(* ---------------------------------------------------------------------------
Func name   : 	Off
Description : 	Sets the Indicator output to FALSE.
Inputs      :	None
Returns     : 	None
Notes       : 	
--------------------------------------------------------------------------- *)

METHOD Off
VAR_INPUT
END_VAR
m_signal^ := FALSE;
END_METHOD

(* ---------------------------------------------------------------------------
Func name   : 	On
Description : 	Sets the Indicator output to TRUE.
Inputs      :	None
Returns     : 	None
Notes       : 	
--------------------------------------------------------------------------- *)

METHOD On
VAR_INPUT
END_VAR
m_signal^ := TRUE;
END_METHOD

END_FUNCTION_BLOCK

// 20 Program Organization Units/Instrument-Controller Functions/fb_STARTP_ControlActuator
(*UPDATE: 			October. 29 2020 - Graham Hunter
					This function block converts a Real Signal/Command to a 4-20 mA signal to be processed by fb_AnalogOutputActuator.
					(Most of the functionality was duplicated from fb_ENDP_Analog but instead of converting a 4-20 mA signal to a Physical Signal, it converts a Physical Signal/Command to a 4-20 mA signal.)
*)

(*UPDATE: 			March. 18 2021 - Jaison Schaab

					Code Ported from Wago.
					
					Code has NOT Yet been tested.
*)

FUNCTION_BLOCK fb_STARTP_ControlActuator
VAR_INPUT
	PhysicalSignal 		: REAL; // this is a physical signal like speed
END_VAR
VAR_OUTPUT
	AnalogSignalValue   : REAL; // this is a 4-20 mA signal
	endpState : INT;
END_VAR
VAR
	m_pActuator420 : POINTER TO fb_AnalogOutputActuator;
	m_inMin 	: REAL;
	m_inMax 	: REAL;
	m_outMin 	: REAL;
	m_outMax 	: REAL;
	m_outpdiffMultiplier 	: REAL;
	m_inpdiffDivisor 		: REAL;
	m_offset 		: REAL;
	m_hysteresis 	: REAL;
	//this is all alarm-related down from here. Should be separated into Alarmable interface, if possible.
	m_devId					: UDeviceId;			// Device Id used for alarm integration
	//m_pAlarmHandler : POINTER TO fb_AlarmHandler; //Alarm handler function pointer
	LowAlarmMonitor 		: fb_AlarmMonitor;
	LowWarningMonitor 		: fb_AlarmMonitor;
	HighWarningMonitor 		: fb_AlarmMonitor;
	HighAlarmMonitor 		: fb_AlarmMonitor;
END_VAR
VAR CONSTANT
	DELAY_TON	: TIME := T#200MS;	//AlarmMonitor delay for Value to DEFINITEVILY cross the alarm limit boundary. and then Trigger.
END_VAR

//get transducers Value scaled from Physical to 4-20 
AnalogSignalValue := Scale(PhysicalSignal);

// None of the below is used currently on the 750-563 card currently <GRAHAM>
//Monitor alarms.
//LowAlarmMonitor.MonitorReal(AnalogSignalValue);
//LowWarningMonitor.MonitorReal(AnalogSignalValue);
//HighWarningMonitor.MonitorReal(AnalogSignalValue);
//HighAlarmMonitor.MonitorReal(AnalogSignalValue);

//ALSO_ update the so-called GaugeState. It controls Needle-Color. BY-DESIGN HW-Error also paints Needle in RED.

(* ---------------------------------------------------------------------------
Func name   : 	FB_init
Description : 	ENDP_Analog_Actuator
Inputs      :	4 reals - Two real values are the input range of the Physical Signal and Two real values are the output range of the Analog Signal.  
Returns     : 	None
--------------------------------------------------------------------------- *)

METHOD FB_init : BOOL
VAR_INPUT
	bInitRetains 		: BOOL; 		// if TRUE, the retain variables are initialized (warm start / cold start)
    bInCopyCode  		: BOOL; 		// if TRUE, the instance afterwards gets moved into the copy code (online change)
	
	//ptrActuator : POINTER TO fb_AnalogOutputActuator;
	PhysicalMin	: REAL;
	PhysicalMax	: REAL;
	AnalogMin 	: REAL;
	AnalogMax 	: REAL;
	//perctHysteresis : REAL;
END_VAR
//m_pActuator420 := ptrActuator;
m_inMin := PhysicalMin;
m_inMax := PhysicalMax;
m_outMin := AnalogMin;   //these are the range of analog values, 4-20 mA 0-10 VDC etc.
m_outMax := AnalogMax;    //that the physical signal is scaled to.
//m_outMin := m_pActuator420^.GetMinInput;   //these are the range of analog values, 4-20 mA 0-10 VDC etc.
//m_outMax := m_pActuator420^.GetMaxInput;    //that the physical signal is scaled to.
m_outpdiffMultiplier := (m_outMax - m_outMin);
m_inpdiffDivisor := (m_inMax - m_inMin);
IF (0.0 = m_inpdiffDivisor) THEN
	m_inpdiffDivisor := 0.000001; //protect against div-by-0, only ONCE, and produce VERY-LARGE Bad value.
                                  //Beckhoff-tcNov was doing this A.every cycle and B.returned 0.0 if Bad, which is normal value. hard to notice.
END_IF

//m_pAlarmHandler := ADR(gAlarmHandler); //i am no longer handling Alarms myself. AlarmMonitor does interfacing to 'gAlarmHandler'.
//m_devId := m_pTxducer420^.GetDevId();

//m_hysteresis := perctHysteresis/100;
//LowAlarmMonitor.Init(f_AlarmCode(m_devId, f_FaultCode(TFaultPriority.Warning, TFaultCondition.UnderLimit)), TAlarmMonitorType.lower_limit, DELAY_TON);
//LowWarningMonitor.Init(f_AlarmCode(m_devId, f_FaultCode(TFaultPriority.Warning, TFaultCondition.UnderWarning)), TAlarmMonitorType.lower_limit, DELAY_TON);
//HighWarningMonitor.Init(f_AlarmCode(m_devId, f_FaultCode(TFaultPriority.Warning, TFaultCondition.OverWarning)), TAlarmMonitorType.upper_limit, DELAY_TON);
//HighAlarmMonitor.Init(f_AlarmCode(m_devId, f_FaultCode(TFaultPriority.Warning, TFaultCondition.OverLimit)), TAlarmMonitorType.upper_limit, DELAY_TON);
END_METHOD

(* ---------------------------------------------------------------------------
Func name   : 	GetConfigData
Description : 	equivalent of "Configure" bkhff-legacy-names.
				
Inputs      :	2-end-range-values, 1 offset, 4 alarms - 7 values.
				state	-	state of the fault
Returns     : 	None
Notes       : 	
--------------------------------------------------------------------------- *)

METHOD GetConfigData
VAR_INPUT
	//cfg : TEndpAnalogCfg;
MinValue : REAL;
MaxValue : REAL;
OffsetValue : REAL;
END_VAR
m_outMin := MinValue;
m_outMax := MaxValue;
m_offset := OffsetValue;
END_METHOD

METHOD GetRange_MinMax
VAR_OUTPUT
	outMinVal : REAL;
	outMaxVal : REAL;
END_VAR
// these are the STARTP product values, in ANALOG UNITS
outMinVal := m_outMin;
outMaxVal := m_outMax;
END_METHOD

METHOD Scale : REAL
VAR_INPUT
	val_mamp : REAL;
END_VAR
Scale := (val_mamp - m_inMin)*m_outpdiffMultiplier/m_inpdiffDivisor + m_outMin;
END_METHOD

METHOD Set_Hysteresis
VAR_INPUT
	perctHysteresis : REAL;
END_VAR
m_hysteresis := perctHysteresis/100;
END_METHOD

METHOD SetRange_MinMax
VAR_INPUT
	AnalogMin : REAL;
	AnalogMax : REAL;
END_VAR
// these are the STARTP product values, in ANALOG Units <GRAHAM>
m_outMin := AnalogMin;
m_outMax := AnalogMax;
END_METHOD

END_FUNCTION_BLOCK

// 20 Program Organization Units/Instrument-Controller Functions/fb_Switch
(*AUTHOR:			Jaison Schaab*)
(*DATE:				March 27 / 2020*)
(*DESCRIPTION: 		This Function Block provides a standard conrol interface for digital
					inputs of type BOOL which includes a debounce feature.*)

(*UPDATE: 			March. 23 2021 - Jaison Schaab

					Code Is fully tested and functional.				
*)

(*UPDATE: 			March. 18 2021 - Jaison Schaab

					Code Ported from Wago.
					
					Code has NOT Yet been tested.
*)

(*UPDATE: 			September. 22 2020 - Jaison Schaab

					Updated the Equals routine to use a bistable block and second falling
					edge timer to now delay the falling edge of the input signal as well
					as the rising edge.
*)	

FUNCTION_BLOCK fb_Switch
VAR_INPUT
END_VAR
VAR_OUTPUT
END_VAR
VAR
	m_pSignal			: POINTER TO BOOL;	// Pointer to the input BOOL signal value
	m_debounce			: TIME;				// Debounce TIME value used for FALSE -> TRUE transition
	m_risingDelayTimer	: TON;				// Debounce timer used for FALSE -> TRUE transition
	m_fallingDelayTimer	: TON;				// Debounce timer used for TRUE -> FALSE transition
	m_signal			: RS;				// Output signal bistable block
END_VAR

(* ---------------------------------------------------------------------------
Func name   : 	Equals
Description : 	Retrieves the current switch value.
Inputs      :	None
Returns     : 	None
Notes       : 	This block is meant to be called cyclically to obtain the
				debounced value, there is no way to override operators in ST.
				
				The signal is delayed on both a FALSE -> TRUE transition
				and a TRUE -> FALSE transition.
--------------------------------------------------------------------------- *)

METHOD Equals : BOOL
VAR_INPUT
END_VAR
// use a rising edge delay timer to debounce the signal on a FALSE -> TRUE transition
m_risingDelayTimer(IN:= m_pSignal^, PT:= m_debounce, Q=> );

// use a falling edge delay timer to debounce the signal on a TRUE -> FALSE transition
m_fallingDelayTimer(IN:= NOT m_pSignal^, PT:= m_debounce, Q=> );

// Output the signal value
m_signal(SET:= m_risingDelayTimer.Q, RESET1:= m_fallingDelayTimer.Q, Q1=> Equals);
END_METHOD

(* ---------------------------------------------------------------------------
Func name   : 	FB_exit
Description : 	Destructor
Inputs      :	None
Returns     : 	None
Notes       : 	
--------------------------------------------------------------------------- *)

METHOD FB_exit : BOOL
VAR_INPUT
	bInCopyCode : BOOL; // if TRUE, the exit method is called for exiting an instance that is copied afterwards (online change)
END_VAR
// Do Nothing
END_METHOD

(* ---------------------------------------------------------------------------
Func name   : 	FB_init
Description : 	Constructor
Inputs      :	signal		-	Pointer to the input BOOL signal value
				debounce	-	Default debounce value of type TIME
Returns     : 	None
Notes       : 	
--------------------------------------------------------------------------- *)

METHOD FB_init : BOOL
VAR_INPUT
	bInitRetains 		: BOOL; 			// if TRUE, the retain variables are initialized (warm start / cold start)
    bInCopyCode  		: BOOL; 			// if TRUE, the instance afterwards gets moved into the copy code (online change)
	signal				: POINTER TO BOOL;	// Pointer to input BOOL signal value 
	debounce			: TIME := T#100MS;	// Default debounce value, can be overridden with Set routine
END_VAR
// Set the local signal pointer
m_pSignal := signal;

// Set the local debounce value to the default value
m_debounce := debounce;
END_METHOD

(* ---------------------------------------------------------------------------
Func name   : 	GetDebounce
Description : 	Gets the debounce time for the switch used to delay the
				the FALSE -> TRUE transition.
Inputs      :	None
Returns     : 	TIME	-	debounce TIME value
Notes       : 	
--------------------------------------------------------------------------- *)

METHOD GetDebounce : TIME
VAR_INPUT
END_VAR
GetDebounce := m_debounce;
END_METHOD

(* ---------------------------------------------------------------------------
Func name   : 	SetDebounce
Description : 	Sets the debounce time for the switch used to delay the
				the FALSE -> TRUE transition.
Inputs      :	debounce	- 	debounce TIME value
Returns     : 	None
Notes       : 	
--------------------------------------------------------------------------- *)

METHOD SetDebounce
VAR_INPUT
	debounce	: TIME;
END_VAR
m_debounce := debounce;
END_METHOD

END_FUNCTION_BLOCK

// 20 Program Organization Units/Interlock Functions/fb_NOVInterlock
(*AUTHOR:		Graham Hunter *)
(*DATE:			Feb 4, 2021 *)
(*DESCRIPTION:	Interlock logic block which interfaces with the NOV and NSA safety interlock PLC*)

(*NOTES:  

INPUTS: 	   Interface consists of external 13 interlock bit inputs and 15 interlock bit cmd override inputs (13 individual interlock override bits, one bypass All override bit, 
			   and one Bypass None Override bit). The Bypass All override supersedes all individual interlock bit overrides as well as the Bypass None override. 
			   The Bypass None override supersedes the individual interlock bit overrides. 
					
VAR_IN_OUTs:   The Function block takes in a VAR_IN_OUT process data structure of the THMINOVInterlock type (from the HMI) that consists of a interlock bit override input WORD (future use) 
			   as well as processed interlock bit output WORD.  
					
FUNCTIONALITY: This function block takes raw external individual interlock bit as inputs and with external individual override bits where one can override single individual interlock bits  
			   or bypass all the individual interlock bits or none of them. The override functionality can be done by the VAR_IN_OUT process data structure as well (in future use).
			   The seperate Process interlock Output word (in future use) will have the status for the individual processed interlock bits as well as status for the overall interlock with bypasses activated or 
			   bypasses not activated.
				  
OUTPUTS:      The output consists of individual processed interlock bits as well as overall status of the interlock block consisting of one ProcessedIntlkOK with No Bypasses bit and one
			  ProcessedIntlkOK with Bypasses. These output bits are fed into the VAR_IN_OUT process data structure.
	  
SIDE NOTE: 
			 Individual processed interlocks are TRUE = (INTLK IS TRUE OR OVERRIDE IS TRUE IF INDIVIDUAL OVERRIDE IS ACTIVE OR BYPASS ALL IS ACTIVE, 
												 FALSE = (INTLK IS FALSE AND OVERRIDE IS FALSE IF INDIVIDUAL OVERRIDE IS INACTIVE OR BYPASS ALL IS INACTIVE)
													
			 IF BYPASS NONE IS ACTIVE & BYPASS ALL IS INACTIVE then     
					processed interlocks are TRUE = (INTLK IS TRUE) 
											 FALSE = (INTLK IS FALSE)
			Note, BYPASS ALL Supersedes BYPASS NONE.
				
EXAMPLE CASE: If one has 3 interlocks out of the 13 used then set the other 10 non-used interlock bits to TRUE and the non-used overrides to FALSE (initially always set to FALSE). 
			  The Bypass All and Bypass None inputs commands can be used on the control engineers discretion.		
	*)
	
(* UPDATE:		April 22, 2021 - Graham Hunter

				Commented out a portion of the Interlock Processing code to be able to mimic NSA interlock logic where m_ProcessedIntlkOKWithBypass is True 
				with just the interlocks being satisfied without any overrides.
				
				Uncommented out the InitAlarms Method that initialize the alarms for when m_ProcessedIntlkOKWithBypass goes from True to False.
				Commented out the m_InterlocksOKAlarm.MonitorBool(value:= m_ProcessedIntlkOKWithBypass) code in fb_NOVInterlock. This code is not passed up as an output yet.
*)

FUNCTION_BLOCK fb_NOVInterlock
VAR_INPUT
	xEnable							: BOOL;
	//stInputData					: TNOVInterlockIn; // Not used as a seperate input from a external device currently, for future use <GRAHAM>
	Intlk01							: BOOL;	// TRUE = (INTLK SATISFIED), FALSE = (INTLK NOT SATISFIED)
	Intlk02							: BOOL;	
	Intlk03							: BOOL;	
	Intlk04							: BOOL;	
	Intlk05							: BOOL;	
	Intlk06							: BOOL;	
	Intlk07							: BOOL;	
	Intlk08							: BOOL;	
	Intlk09							: BOOL;	
	Intlk10							: BOOL;	
	Intlk11 						: BOOL;	
	Intlk12							: BOOL;	
	Intlk13							: BOOL;

	IntlkBypassALL					: BOOL;	// Bypass/override all interlocks command input
	Intlk01Bypass					: BOOL;	// TRUE = (OVERRIDE ACTIVE), FALSE = (OVERRIDE NOT ACTIVE)
	Intlk02Bypass					: BOOL;	
	Intlk03Bypass					: BOOL;	
	Intlk04Bypass					: BOOL;	
	Intlk05Bypass					: BOOL;	
	Intlk06Bypass					: BOOL;	
	Intlk07Bypass					: BOOL;	
	Intlk08Bypass					: BOOL;	
	Intlk09Bypass					: BOOL;	
	Intlk10Bypass					: BOOL;	
	Intlk11Bypass 					: BOOL;	
	Intlk12Bypass					: BOOL;	
	Intlk13Bypass					: BOOL;
	IntlkBypassNONE					: BOOL;	// Do not Bypass/override any interlocks command input	
END_VAR
VAR_OUTPUT
	//stOutputData					: TNOVInterlockStatusOut; // Possible future use of a seperate output WORD
	ProcessedIntlkOK_NoBypass		: BOOL;	// All interlocks are Ok with no bypasses/overrides
	ProcessedIntlk01				: BOOL;	// TRUE = (INTLK IS TRUE OR OVERRIDE IS TRUE IF OVERRIDE IS ACTIVE, FALSE = (INTLK IS FALSE AND OVERRIDE IS FALSE IF OVERRIDE IS ACTIVE)
	ProcessedIntlk02				: BOOL;	
	ProcessedIntlk03				: BOOL;	
	ProcessedIntlk04				: BOOL;	
	ProcessedIntlk05				: BOOL;	
	ProcessedIntlk06				: BOOL;	
	ProcessedIntlk07				: BOOL;	
	ProcessedIntlk08				: BOOL;	
	ProcessedIntlk09				: BOOL;	
	ProcessedIntlk10				: BOOL;	
	ProcessedIntlk11 				: BOOL;	
	ProcessedIntlk12				: BOOL;	
	ProcessedIntlk13				: BOOL;	
	ProcessedIntlkOK_WithBypass		: BOOL;	// All interlocks are Ok with bypasses/overrides
END_VAR
VAR_IN_OUT
	stProcessData					: THMINOVInterlock;	// Possible future use of a DynIn Bypass Cmd status input word
							
END_VAR

VAR
	
// Internal variables
// Internal Inputs
	// Interlock Status
	// Raw Unprocessed Interlocks from NOV or NSA interlocks 
	m_StatusIntlk01				: BOOL;					// TRUE = (INTLK SATISFIED), FALSE = (INTLK NOT SATISFIED)
	m_StatusIntlk02				: BOOL;					// TRUE = (INTLK SATISFIED), FALSE = (INTLK NOT SATISFIED)
	m_StatusIntlk03				: BOOL;					// TRUE = (INTLK SATISFIED), FALSE = (INTLK NOT SATISFIED)
	m_StatusIntlk04				: BOOL;					// TRUE = (INTLK SATISFIED), FALSE = (INTLK NOT SATISFIED)
	m_StatusIntlk05				: BOOL;					// TRUE = (INTLK SATISFIED), FALSE = (INTLK NOT SATISFIED)
	m_StatusIntlk06				: BOOL;					// TRUE = (INTLK SATISFIED), FALSE = (INTLK NOT SATISFIED)
	m_StatusIntlk07				: BOOL;					// TRUE = (INTLK SATISFIED), FALSE = (INTLK NOT SATISFIED)
	m_StatusIntlk08				: BOOL;					// TRUE = (INTLK SATISFIED), FALSE = (INTLK NOT SATISFIED)
	m_StatusIntlk09				: BOOL;					// TRUE = (INTLK SATISFIED), FALSE = (INTLK NOT SATISFIED)
	m_StatusIntlk10				: BOOL;					// TRUE = (INTLK SATISFIED), FALSE = (INTLK NOT SATISFIED)
	m_StatusIntlk11				: BOOL;					// TRUE = (INTLK SATISFIED), FALSE = (INTLK NOT SATISFIED)
	m_StatusIntlk12				: BOOL;					// TRUE = (INTLK SATISFIED), FALSE = (INTLK NOT SATISFIED)
	m_StatusIntlk13				: BOOL;					// TRUE = (INTLK SATISFIED), FALSE = (INTLK NOT SATISFIED)
	m_StatusNoBypassIntlkOK		: BOOL;					// TRUE = Interlocks OK (No Bypasses)
	m_StatusBypassIntlkOK		: BOOL;					// TRUE = Interlocks OK (With Bypasses)
	
	// Function Block Command Input
	m_BlockEnable					: BOOL;				// TRUE = Function Block is Active, FALSE = Inactive
	
	// Bypasses/Override input commands from HMI
	m_BypassCmdIntlkBypassALL		: BOOL;				// Bypass/override all interlocks command input	
	m_BypassCmdIntlk01				: BOOL;				// TRUE = (OVERRIDE ACTIVE), FALSE = (OVERRIDE NOT ACTIVE)
	m_BypassCmdIntlk02				: BOOL;				// TRUE = (OVERRIDE ACTIVE), FALSE = (OVERRIDE NOT ACTIVE)
	m_BypassCmdIntlk03				: BOOL;				// TRUE = (OVERRIDE ACTIVE), FALSE = (OVERRIDE NOT ACTIVE)
	m_BypassCmdIntlk04				: BOOL;				// TRUE = (OVERRIDE ACTIVE), FALSE = (OVERRIDE NOT ACTIVE)
	m_BypassCmdIntlk05				: BOOL;				// TRUE = (OVERRIDE ACTIVE), FALSE = (OVERRIDE NOT ACTIVE)
	m_BypassCmdIntlk06				: BOOL;				// TRUE = (OVERRIDE ACTIVE), FALSE = (OVERRIDE NOT ACTIVE)
	m_BypassCmdIntlk07				: BOOL;				// TRUE = (OVERRIDE ACTIVE), FALSE = (OVERRIDE NOT ACTIVE)
	m_BypassCmdIntlk08				: BOOL;				// TRUE = (OVERRIDE ACTIVE), FALSE = (OVERRIDE NOT ACTIVE)
	m_BypassCmdIntlk09				: BOOL;				// TRUE = (OVERRIDE ACTIVE), FALSE = (OVERRIDE NOT ACTIVE)
	m_BypassCmdIntlk10				: BOOL;				// TRUE = (OVERRIDE ACTIVE), FALSE = (OVERRIDE NOT ACTIVE)
	m_BypassCmdIntlk11				: BOOL;				// TRUE = (OVERRIDE ACTIVE), FALSE = (OVERRIDE NOT ACTIVE)
	m_BypassCmdIntlk12				: BOOL;				// TRUE = (OVERRIDE ACTIVE), FALSE = (OVERRIDE NOT ACTIVE)
	m_BypassCmdIntlk13				: BOOL;				// TRUE = (OVERRIDE ACTIVE), FALSE = (OVERRIDE NOT ACTIVE)
	m_BypassCmdIntlkBypassNONE		: BOOL;				// Do not Bypass/override any interlocks command input
	
	
// Internal Outputs
	// Processed Interlocks
	m_ProcessedIntlkOKNoBypass	: BOOL;					// All interlocks are Ok with no bypasses/overrides
	m_ProcessedIntlk01			: BOOL;					// TRUE = (INTLK IS TRUE OR OVERRIDE IS TRUE), FALSE = (INTLK IS FALSE AND OVERRIDE IS FALSE)
	m_ProcessedIntlk02			: BOOL;						
	m_ProcessedIntlk03			: BOOL;						
	m_ProcessedIntlk04			: BOOL;						
	m_ProcessedIntlk05			: BOOL;						
	m_ProcessedIntlk06			: BOOL;						
	m_ProcessedIntlk07			: BOOL;						
	m_ProcessedIntlk08			: BOOL;						
	m_ProcessedIntlk09			: BOOL;						
	m_ProcessedIntlk10			: BOOL;						
	m_ProcessedIntlk11			: BOOL;						
	m_ProcessedIntlk12			: BOOL;						
	m_ProcessedIntlk13			: BOOL;						
	m_ProcessedIntlkOKWithBypass: BOOL;					// All interlocks are Ok with bypasses/overrides
	
	// Fault Handling (Alarms)
	m_devId							: UDeviceId;		// Device Id used for alarm integration
	
// Alarms
	
	m_InterlocksOKAlarm				: fb_AlarmMonitor;	// Alarm monitor for interlock conditions, Alarm is SET if ANY interlock condition is not met
	
END_VAR

// Cycle Inputs
// Update Controls
m_BlockEnable := xEnable;					// Enable the Interlock block logic when this block is enabled

IF m_BlockEnable THEN

// Cycle Var_in_out Inputs

// Bypass Input Commands from HMI, Cycle Var_in_out Inputs, A little dangerous to not be able to see the active HMIInterlock bypasses when calling this FB <GRAHAM>
// Bypass Input Commands from HMI commented out for now, for future use, HMI may have the ability to override in the future <GRAHAM>
m_BypassCmdIntlkBypassALL		:= (*stProcessData.HMIInterlockBypass.IntlkBypassALL OR*)IntlkBypassALL; // Bypass/override all interlocks command input
m_BypassCmdIntlk01				:= (*stProcessData.HMIInterlockBypass.Intlk01Bypass OR*) Intlk01Bypass;	// TRUE = (OVERRIDE ACTIVE), FALSE = (OVERRIDE NOT ACTIVE)
m_BypassCmdIntlk02				:= (*stProcessData.HMIInterlockBypass.Intlk02Bypass OR*) Intlk02Bypass;	// TRUE = (OVERRIDE ACTIVE), FALSE = (OVERRIDE NOT ACTIVE)
m_BypassCmdIntlk03				:= (*stProcessData.HMIInterlockBypass.Intlk03Bypass OR*) Intlk03Bypass;	// TRUE = (OVERRIDE ACTIVE), FALSE = (OVERRIDE NOT ACTIVE)
m_BypassCmdIntlk04				:= (*stProcessData.HMIInterlockBypass.Intlk04Bypass OR*) Intlk04Bypass;	// TRUE = (OVERRIDE ACTIVE), FALSE = (OVERRIDE NOT ACTIVE)
m_BypassCmdIntlk05				:= (*stProcessData.HMIInterlockBypass.Intlk05Bypass OR*) Intlk05Bypass;	// TRUE = (OVERRIDE ACTIVE), FALSE = (OVERRIDE NOT ACTIVE)
m_BypassCmdIntlk06				:= (*stProcessData.HMIInterlockBypass.Intlk06Bypass OR*) Intlk06Bypass;	// TRUE = (OVERRIDE ACTIVE), FALSE = (OVERRIDE NOT ACTIVE)
m_BypassCmdIntlk07				:= (*stProcessData.HMIInterlockBypass.Intlk07Bypass OR*) Intlk07Bypass;	// TRUE = (OVERRIDE ACTIVE), FALSE = (OVERRIDE NOT ACTIVE)
m_BypassCmdIntlk08				:= (*stProcessData.HMIInterlockBypass.Intlk08Bypass OR*) Intlk08Bypass;	// TRUE = (OVERRIDE ACTIVE), FALSE = (OVERRIDE NOT ACTIVE)
m_BypassCmdIntlk09				:= (*stProcessData.HMIInterlockBypass.Intlk09Bypass OR*) Intlk09Bypass;	// TRUE = (OVERRIDE ACTIVE), FALSE = (OVERRIDE NOT ACTIVE)
m_BypassCmdIntlk10				:= (*stProcessData.HMIInterlockBypass.Intlk10Bypass OR*) Intlk10Bypass;	// TRUE = (OVERRIDE ACTIVE), FALSE = (OVERRIDE NOT ACTIVE)
m_BypassCmdIntlk11				:= (*stProcessData.HMIInterlockBypass.Intlk11Bypass OR*) Intlk11Bypass;	// TRUE = (OVERRIDE ACTIVE), FALSE = (OVERRIDE NOT ACTIVE)
m_BypassCmdIntlk12				:= (*stProcessData.HMIInterlockBypass.Intlk12Bypass OR*) Intlk12Bypass;	// TRUE = (OVERRIDE ACTIVE), FALSE = (OVERRIDE NOT ACTIVE)
m_BypassCmdIntlk13				:= (*stProcessData.HMIInterlockBypass.Intlk13Bypass OR*) Intlk13Bypass;	// TRUE = (OVERRIDE ACTIVE), FALSE = (OVERRIDE NOT ACTIVE)
m_BypassCmdIntlkBypassNONE		:= (*stProcessData.HMIInterlockBypass.IntlkBypassNONE OR*) IntlkBypassNONE; // Do not Bypass/override any interlocks command input

// Raw Unprocessed Interlocks from NOV or NSA
m_StatusIntlk01				:= Intlk01;		// TRUE = (INTLK SATISFIED), FALSE = (INTLK NOT SATISFIED)
m_StatusIntlk02				:= Intlk02;			
m_StatusIntlk03				:= Intlk03;			
m_StatusIntlk04				:= Intlk04;			
m_StatusIntlk05				:= Intlk05;			
m_StatusIntlk06				:= Intlk06;			
m_StatusIntlk07				:= Intlk07;			
m_StatusIntlk08				:= Intlk08;			
m_StatusIntlk09				:= Intlk09;			
m_StatusIntlk10				:= Intlk10;			
m_StatusIntlk11				:= Intlk11;			
m_StatusIntlk12				:= Intlk12;			
m_StatusIntlk13				:= Intlk13;	

//// Interlock Processing Code START
// Process the Interlock Bits
IF NOT m_BypassCmdIntlkBypassALL THEN
	IF m_BypassCmdIntlkBypassNONE THEN
		
		m_ProcessedIntlkOKNoBypass := m_StatusIntlk01 AND m_StatusIntlk02 AND m_StatusIntlk03 AND m_StatusIntlk04 AND m_StatusIntlk05 AND m_StatusIntlk06
									  AND m_StatusIntlk07 AND m_StatusIntlk08 AND m_StatusIntlk09 AND m_StatusIntlk10 AND m_StatusIntlk11 AND m_StatusIntlk12 AND m_StatusIntlk13;
		m_ProcessedIntlk01 := m_StatusIntlk01; // TRUE = (INTLK IS TRUE), FALSE = (INTLK IS FALSE), RAW INTERLOCKS WITHOUT OVERRIDES
		m_ProcessedIntlk02 := m_StatusIntlk02;
		m_ProcessedIntlk03 := m_StatusIntlk03;
		m_ProcessedIntlk04 := m_StatusIntlk04;
		m_ProcessedIntlk05 := m_StatusIntlk05;
		m_ProcessedIntlk06 := m_StatusIntlk06;
		m_ProcessedIntlk07 := m_StatusIntlk07;
		m_ProcessedIntlk08 := m_StatusIntlk08;
		m_ProcessedIntlk09 := m_StatusIntlk09;
		m_ProcessedIntlk10 := m_StatusIntlk10;
		m_ProcessedIntlk11 := m_StatusIntlk11;
		m_ProcessedIntlk12 := m_StatusIntlk12;
		m_ProcessedIntlk13 := m_StatusIntlk13;
		m_ProcessedIntlkOKWithBypass := FALSE;
		(*m_ProcessedIntlkOKWithBypass := m_StatusIntlk01 AND m_StatusIntlk02 AND m_StatusIntlk03 AND m_StatusIntlk04 AND m_StatusIntlk05 AND m_StatusIntlk06
									  AND m_StatusIntlk07 AND m_StatusIntlk08 AND m_StatusIntlk09 AND m_StatusIntlk10 AND m_StatusIntlk11 AND m_StatusIntlk12 AND m_StatusIntlk13; 
		// interlocks may be OK regardless of Bypass/Override not being active*)
						  					  
	ELSIF NOT m_BypassCmdIntlkBypassNONE THEN
		
		m_ProcessedIntlkOKNoBypass := m_StatusIntlk01 AND m_StatusIntlk02 AND m_StatusIntlk03 AND m_StatusIntlk04 AND m_StatusIntlk05 AND m_StatusIntlk06
									  AND m_StatusIntlk07 AND m_StatusIntlk08 AND m_StatusIntlk09 AND m_StatusIntlk10 AND m_StatusIntlk11 AND m_StatusIntlk12 AND m_StatusIntlk13;
		m_ProcessedIntlk01 := m_StatusIntlk01 OR m_BypassCmdIntlk01; // TRUE = (INTLK IS TRUE OR INTLK OVERRIDE IS TRUE), FALSE = (INTLK IS FALSE AND INTLK OVERRIDE IS FALSE)
		m_ProcessedIntlk02 := m_StatusIntlk02 OR m_BypassCmdIntlk02;
		m_ProcessedIntlk03 := m_StatusIntlk03 OR m_BypassCmdIntlk03;
		m_ProcessedIntlk04 := m_StatusIntlk04 OR m_BypassCmdIntlk04;
		m_ProcessedIntlk05 := m_StatusIntlk05 OR m_BypassCmdIntlk05;
		m_ProcessedIntlk06 := m_StatusIntlk06 OR m_BypassCmdIntlk06;
		m_ProcessedIntlk07 := m_StatusIntlk07 OR m_BypassCmdIntlk07;
		m_ProcessedIntlk08 := m_StatusIntlk08 OR m_BypassCmdIntlk08;
		m_ProcessedIntlk09 := m_StatusIntlk09 OR m_BypassCmdIntlk09;
		m_ProcessedIntlk10 := m_StatusIntlk10 OR m_BypassCmdIntlk10;
		m_ProcessedIntlk11 := m_StatusIntlk11 OR m_BypassCmdIntlk11;
		m_ProcessedIntlk12 := m_StatusIntlk12 OR m_BypassCmdIntlk12;
		m_ProcessedIntlk13 := m_StatusIntlk13 OR m_BypassCmdIntlk13;
		(*IF m_BypassCmdIntlk01 OR m_BypassCmdIntlk02 OR m_BypassCmdIntlk03 OR m_BypassCmdIntlk04 OR m_BypassCmdIntlk05 OR m_BypassCmdIntlk06 OR 
		   m_BypassCmdIntlk07 OR m_BypassCmdIntlk08 OR m_BypassCmdIntlk09 OR m_BypassCmdIntlk10 OR m_BypassCmdIntlk11 OR m_BypassCmdIntlk12 OR m_BypassCmdIntlk13 THEN*)
			m_ProcessedIntlkOKWithBypass := (m_StatusIntlk01 OR m_BypassCmdIntlk01) AND (m_StatusIntlk02 OR m_BypassCmdIntlk02) AND (m_StatusIntlk03 OR m_BypassCmdIntlk03) 
											AND (m_StatusIntlk04 OR m_BypassCmdIntlk04) AND (m_StatusIntlk05 OR m_BypassCmdIntlk05) AND (m_StatusIntlk06 OR m_BypassCmdIntlk06)
											AND (m_StatusIntlk07 OR m_BypassCmdIntlk07) AND (m_StatusIntlk08 OR m_BypassCmdIntlk08) AND (m_StatusIntlk09 OR m_BypassCmdIntlk09) 
											AND (m_StatusIntlk10 OR m_BypassCmdIntlk10) AND (m_StatusIntlk11 OR m_BypassCmdIntlk11) AND (m_StatusIntlk12 OR m_BypassCmdIntlk12)
											AND (m_StatusIntlk13 OR m_BypassCmdIntlk13);
		(*ELSE
			m_ProcessedIntlkOKWithBypass := FALSE;
			
		END_IF*)
		// Commented out the above code to be able to mimic NSA interlock logic where m_ProcessedIntlkOKWithBypass is True with just the interlocks being satisfied without any overrides, 04/07/2021 <GRAHAM> 	 						
	END_IF
		
ELSIF m_BypassCmdIntlkBypassALL THEN
	
	m_ProcessedIntlkOKNoBypass := FALSE;
	m_ProcessedIntlk01 := TRUE; // TRUE = ALL INTERLOCKS OVERRIDDEN
	m_ProcessedIntlk02 := TRUE;
	m_ProcessedIntlk03 := TRUE;
	m_ProcessedIntlk04 := TRUE;
	m_ProcessedIntlk05 := TRUE;
	m_ProcessedIntlk06 := TRUE;
	m_ProcessedIntlk07 := TRUE;
	m_ProcessedIntlk08 := TRUE;
	m_ProcessedIntlk09 := TRUE;
	m_ProcessedIntlk10 := TRUE;
	m_ProcessedIntlk11 := TRUE;
	m_ProcessedIntlk12 := TRUE;
	m_ProcessedIntlk13 := TRUE;
	m_ProcessedIntlkOKWithBypass := TRUE; //TRUE = ALL INTERLOCKS OVERRIDDEN
	
END_IF
//// Interlock Processing Code END


// Output the current interlock status variables

// Update Alarms
// m_InterlocksOKAlarm.MonitorBool(value			:= m_ProcessedIntlkOKWithBypass);	// Triggers alarm when FALSE

// Cycle Outputs
(* Possible future use of seperate output WORD out of the function block
stOutputData.InterlockProcessed.IntlkOK_NoBypass := m_ProcessedIntlkOKNoBypass; // All interlocks are Ok with no bypasses/overrides
stOutputData.InterlockProcessed.Intlk01:= m_ProcessedIntlk01; 					// TRUE = (INTLK IS TRUE OR OVERRIDE IS TRUE IF OVERRIDE IS ACTIVE, FALSE = (INTLK IS FALSE AND OVERRIDE IS FALSE IF OVERRIDE IS ACTIVE)
stOutputData.InterlockProcessed.Intlk02:= m_ProcessedIntlk02;
stOutputData.InterlockProcessed.Intlk03:= m_ProcessedIntlk03;
stOutputData.InterlockProcessed.Intlk04:= m_ProcessedIntlk04;
stOutputData.InterlockProcessed.Intlk05:= m_ProcessedIntlk05;
stOutputData.InterlockProcessed.Intlk06:= m_ProcessedIntlk06;
stOutputData.InterlockProcessed.Intlk07:= m_ProcessedIntlk07;
stOutputData.InterlockProcessed.Intlk08:= m_ProcessedIntlk08;
stOutputData.InterlockProcessed.Intlk09:= m_ProcessedIntlk09;
stOutputData.InterlockProcessed.Intlk10:= m_ProcessedIntlk10;
stOutputData.InterlockProcessed.Intlk11:= m_ProcessedIntlk11;
stOutputData.InterlockProcessed.Intlk12:= m_ProcessedIntlk12;
stOutputData.InterlockProcessed.Intlk13:= m_ProcessedIntlk13;
stOutputData.InterlockProcessed.IntlkOK_WithBypass:= m_ProcessedIntlkOKWithBypass;*)

ProcessedIntlkOK_NoBypass		:= m_ProcessedIntlkOKNoBypass;	// All interlocks are Ok with no bypasses/overrides
ProcessedIntlk01				:= m_ProcessedIntlk01;			// TRUE = (INTLK IS TRUE OR OVERRIDE IS TRUE IF OVERRIDE IS ACTIVE, FALSE = (INTLK IS FALSE AND OVERRIDE IS FALSE IF OVERRIDE IS ACTIVE)
ProcessedIntlk02				:= m_ProcessedIntlk02;	
ProcessedIntlk03				:= m_ProcessedIntlk03;	
ProcessedIntlk04				:= m_ProcessedIntlk04;	
ProcessedIntlk05				:= m_ProcessedIntlk05;	
ProcessedIntlk06				:= m_ProcessedIntlk06;	
ProcessedIntlk07				:= m_ProcessedIntlk07;	
ProcessedIntlk08				:= m_ProcessedIntlk08;	
ProcessedIntlk09				:= m_ProcessedIntlk09;	
ProcessedIntlk10				:= m_ProcessedIntlk10;	
ProcessedIntlk11 				:= m_ProcessedIntlk11;	
ProcessedIntlk12				:= m_ProcessedIntlk12;	
ProcessedIntlk13				:= m_ProcessedIntlk13;	
ProcessedIntlkOK_WithBypass		:= m_ProcessedIntlkOKWithBypass;// All interlocks are Ok with bypasses/overrides

// Cycle Var_in_out Outputs
// Cycle Var_in_out DynOut Interlock status out word
stProcessData.HMIInterlockProcessed.IntlkOK_NoBypass	 := m_ProcessedIntlkOKNoBypass;
stProcessData.HMIInterlockProcessed.Intlk01 			 := m_ProcessedIntlk01;
stProcessData.HMIInterlockProcessed.Intlk02 			 := m_ProcessedIntlk02;
stProcessData.HMIInterlockProcessed.Intlk03				 := m_ProcessedIntlk03;
stProcessData.HMIInterlockProcessed.Intlk04				 := m_ProcessedIntlk04;
stProcessData.HMIInterlockProcessed.Intlk05 			 := m_ProcessedIntlk05;
stProcessData.HMIInterlockProcessed.Intlk06 			 := m_ProcessedIntlk06;
stProcessData.HMIInterlockProcessed.Intlk07				 := m_ProcessedIntlk07;
stProcessData.HMIInterlockProcessed.Intlk08				 := m_ProcessedIntlk08;
stProcessData.HMIInterlockProcessed.Intlk09 			 := m_ProcessedIntlk09;
stProcessData.HMIInterlockProcessed.Intlk10 			 := m_ProcessedIntlk10;
stProcessData.HMIInterlockProcessed.Intlk11				 := m_ProcessedIntlk11;
stProcessData.HMIInterlockProcessed.Intlk12				 := m_ProcessedIntlk12;
stProcessData.HMIInterlockProcessed.Intlk13				 := m_ProcessedIntlk13;
stProcessData.HMIInterlockProcessed.IntlkOK_WithBypass	 := m_ProcessedIntlkOKWithBypass;

END_IF

/// ---------------------------------------------------------------------------
///Func name   : 	FB_exit
///Description : 	Destructor
///Inputs      :	None
///Returns     : 	None
///Notes       : 	
///--------------------------------------------------------------------------- 
METHOD FB_exit : BOOL
VAR_INPUT
	/// if TRUE, the exit method is called for exiting an instance that is copied afterwards (online change)
	bInCopyCode: BOOL;
END_VAR
// Do nothing
END_METHOD

/// ---------------------------------------------------------------------------
///Func name   : 	FB_init
///Description : 	Constructor
///Inputs      :	None
///Returns     : 	None
///Notes       : 	
///--------------------------------------------------------------------------- 
METHOD FB_init
VAR_INPUT
	bInitRetains: BOOL;
	bInCopyCode: BOOL;
END_VAR
END_METHOD

(* ---------------------------------------------------------------------------
Func name   : 	InitAlarms
Description : 	Initializes the alarm monitors.
Inputs      :	devId	:	Device Id used for alarm integration
Returns     : 	None
Notes       : 	
--------------------------------------------------------------------------- *)

METHOD InitAlarms
VAR_INPUT
	devId		: UDeviceId;	// Device Id used for alarm integration
END_VAR
// Set the device id which is used for alarm integration
m_devId := devId;

// Initialize the alarm monitors and set their limits
m_InterlocksOKAlarm.InitAlarm(code:= f_AlarmCode(devId, f_FaultCode(TFaultPriority.Error, TFaultCondition.Interlock)), alarmType:= TAlarmMonitorType.lower_limit, delayTime:= T#0S);
m_InterlocksOKAlarm.SetLimitBool(on:= FALSE, off:= TRUE);
m_InterlocksOKAlarm.EnableLimit();
END_METHOD

END_FUNCTION_BLOCK

// 20 Program Organization Units/Modbus/fb_ModbusError
(*AUTHOR:			Jaison Schaab*)
(*DATE:				November 5 / 2019*)
(*DESCRIPTION: 		This Function Block calculates if a modbus communication failure has occured
					as defined as 2x the input timeout value.*)

(*UPDATE: 			March. 18 2021 - Jaison Schaab

					Code Ported from Wago.
					
					Code Is fully tested and functional.
*)

FUNCTION_BLOCK fb_ModbusError
VAR_INPUT
	xBusy			: BOOL;
	xError			: BOOL;
	tTimeOut		: TIME;
END_VAR
VAR_OUTPUT
	xFailure		: BOOL;
END_VAR
VAR
	dly				: TON;
	hld				: RS;
END_VAR

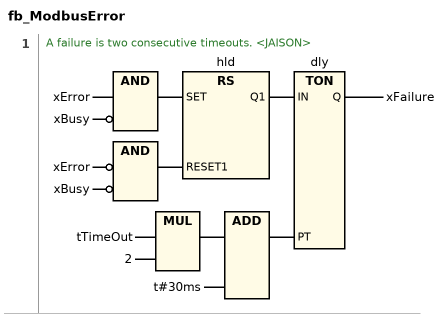
// NETWORK 1
// A failure is two consecutive timeouts. <JAISON>
hld(SET := xError AND NOT xBusy, RESET1 := NOT xError AND NOT xBusy); // RS
dly(IN := hld.Q1, PT := tTimeOut * 2 + t#30ms); // TON
xFailure := dly.Q;

END_FUNCTION_BLOCK

// 20 Program Organization Units/Modbus/fb_ModbusServer
(*AUTHOR:			Jaison Schaab*)
(*DATE:				March 10 / 2021*)
(*DESCRIPTION: 		This Function Block provides a standard data access model to the Modbus TCP Server  (TF6250) 
					whitch is executed seperately as a windows OS service.
*					To access the data simply call the "Get" routines which return pointers (of specified type WORD
*					or BOOL) which can be used to copy the data from/to in order the interact with any connected
*					master stations.*)

(*NOTES:
*
*	In order to use the modbus server the Modbus TCP (TF6250) function must be installed on the PLC as well as be properly licensed.
*	
*	The modbus server runs as a seprate windows OS service and is to interacted with through this class.  In order to properly setup
*	the server it must be configured with the proper NOV configuration XML file using the beckhoff configurator tool.  This XML file
*	is specifically setup for use with the this stdNOV library class and should be found with the library in the revision control system.
*
*	The configurator is installed per default to the directory \TwinCAT3\Functions\TF6250-Modbus-TCP. The tools allow to read and 
*	change the actual configuration of TwinCAT Modbus TCP server.
*
<TODO>
*	Beckhoff support has advised no MAX limit on the number of simultaneous connections.  
*	<TODO> Could be a TCP connection limit? Need to confirm?
*
*)

(*UPDATE: 			March. 18 2021 - Jaison Schaab

					Code Ported from Wago.
					
					Code Is fully tested and functional, however missing the connection list functionality
					previously implimented on the Wago controller.  I am still working with Beckhoff support
					on a solution, perhaps intercepting all TCP packets and filtering them?
*)

FUNCTION_BLOCK fb_ModbusServer
VAR_INPUT
	xEnable							: BOOL;						// Input to enable the Block
	stModbusServer					: TModbusServerConfig;		// Modbus server configuration
END_VAR
VAR_OUTPUT
	xComFailure						: BOOL;						// TRUE if modbus communication is not present (Reads/Writes to server)	
	uiConnectedClients				: UINT;						// Number of server connections -> <FUTURE> connected clients to the server
END_VAR
VAR
	m_GetConnectedClientCount		: ADSREAD;					// ADS READ of the number of connected Modbus clients
	m_udiConnectedClients			: UDINT;					// Internal number of actually connected masters to the server
		
	m_GetModbusRequestCount			: ADSREAD;					// ADS READ of the received Modbus requests
	m_CurrentRequestCount			: UDINT;					// Current scan request counter, used for detecting comm loss
		
	m_GetModbusResponseCount		: ADSREAD;					// ADS READ of the received Modbus answers
	m_CurrentResponseCount			: UDINT;					// Current scan scan response counter, used for detecting comm loss
	
	m_tmrNoComms					: TON;						// Comm loss timer, used to delay setting the comm loss bit
	m_oldRequestCount				: UDINT;					// Memory of previous scan request counter, used for detecting comm loss
	m_oldResponseCount				: UDINT;					// Memory of previous scan response counter, used for detecting comm loss
	
	// List of all connected clients <JAISON>
	m_ConnectionList				: ARRAY[1..MAX_CONNECTIONS] OF TModbusServerConnection;
END_VAR
VAR CONSTANT
	// MAX number of connected clients used for sizing the connected clients array.
	// Default is 20. <JAISON>
	MAX_CONNECTIONS					: INT := 20;
END_VAR

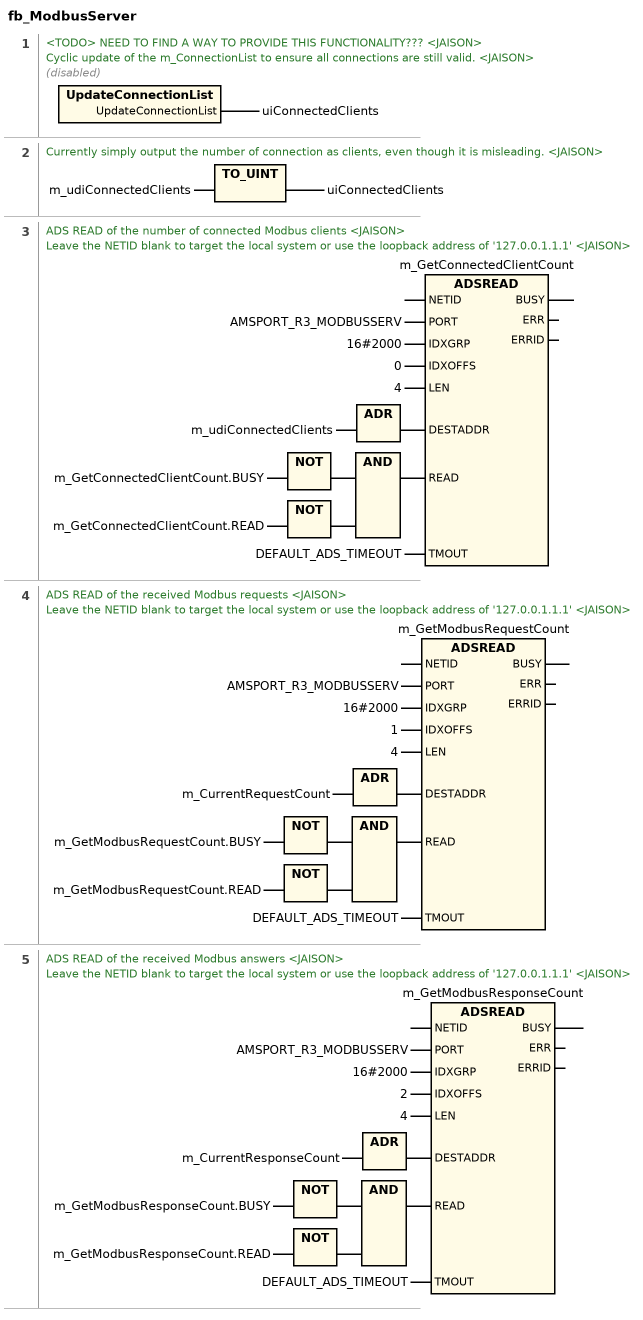
// NETWORK 1 (disabled)
// <TODO> NEED TO FIND A WAY TO PROVIDE THIS FUNCTIONALITY??? <JAISON>
// Cyclic update of the m_ConnectionList to ensure all connections are still valid. <JAISON>
// uiConnectedClients := UpdateConnectionList();

// NETWORK 2
// Currently simply output the number of connection as clients, even though it is misleading. <JAISON>
uiConnectedClients := TO_UINT(m_udiConnectedClients);

// NETWORK 3
// ADS READ of the number of connected Modbus clients <JAISON>
//
// Leave the NETID blank to target the local system or use the loopback address of '127.0.0.1.1.1' <JAISON>
m_GetConnectedClientCount(
    PORT := AMSPORT_R3_MODBUSSERV,
    IDXGRP := 16#2000,
    IDXOFFS := 0,
    LEN := 4,
    DESTADDR := ADR(m_udiConnectedClients),
    READ := NOT m_GetConnectedClientCount.BUSY AND NOT m_GetConnectedClientCount.READ,
    TMOUT := DEFAULT_ADS_TIMEOUT); // ADSREAD

// NETWORK 4
// ADS READ of the received Modbus requests <JAISON>
//
// Leave the NETID blank to target the local system or use the loopback address of '127.0.0.1.1.1' <JAISON>
m_GetModbusRequestCount(
    PORT := AMSPORT_R3_MODBUSSERV,
    IDXGRP := 16#2000,
    IDXOFFS := 1,
    LEN := 4,
    DESTADDR := ADR(m_CurrentRequestCount),
    READ := NOT m_GetModbusRequestCount.BUSY AND NOT m_GetModbusRequestCount.READ,
    TMOUT := DEFAULT_ADS_TIMEOUT); // ADSREAD

// NETWORK 5
// ADS READ of the received Modbus answers <JAISON>
//
// Leave the NETID blank to target the local system or use the loopback address of '127.0.0.1.1.1' <JAISON>
m_GetModbusResponseCount(
    PORT := AMSPORT_R3_MODBUSSERV,
    IDXGRP := 16#2000,
    IDXOFFS := 2,
    LEN := 4,
    DESTADDR := ADR(m_CurrentResponseCount),
    READ := NOT m_GetModbusResponseCount.BUSY AND NOT m_GetModbusResponseCount.READ,
    TMOUT := DEFAULT_ADS_TIMEOUT); // ADSREAD

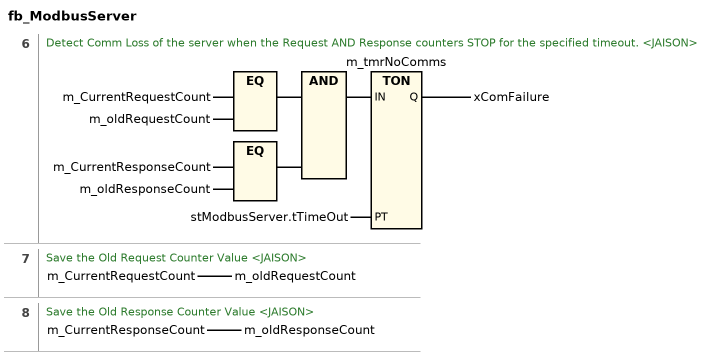
// NETWORK 6
// Detect Comm Loss of the server when the Request AND Response counters STOP for the specified timeout. <JAISON>
m_tmrNoComms(IN := m_CurrentRequestCount = m_oldRequestCount AND m_CurrentResponseCount = m_oldResponseCount, PT := stModbusServer.tTimeOut); // TON
xComFailure := m_tmrNoComms.Q;

// NETWORK 7
// Save the Old Request Counter Value <JAISON>
m_oldRequestCount := m_CurrentRequestCount;

// NETWORK 8
// Save the Old Response Counter Value <JAISON>
m_oldResponseCount := m_CurrentResponseCount;

// NOT IMPLIMENTED FOR BECKHOFF AS IT DOES NOT SUPPORT THIS FUNCTIONALITY <JAISON>

(* ---------------------------------------------------------------------------
Func name   : 	afterAccess
Description : 	Data access listener interface routine for the modbus server
				TCP connection which is called AFTER any access to the modbus
				data model spaces.
Inputs      :	sClientId		-	IP Address of the connected client
				bUnitId			-	Unit id of the requested data model
				bFunctionCode	-	Modbus function code used to access data model
				wReadAddress	-	Address of data model read request
				wReadQuantity	-	Quantity of registers being read (in BOOL or WORD)
				wWriteAddress	-	Address of data model write request
				wWriteQuantity	-	Quantity of registers being written (in BOOL or WORD)
				oStatus			-	Content of a "WagoTypesErrorBase.I_Result" object
Returns     : 	None
Notes       : 	
--------------------------------------------------------------------------- *)

METHOD afterAccess
VAR_INPUT
	sClientId		: STRING(20);	// who is asking
	bUnitId			: BYTE;			// unit id of the requested data model
	bFunctionCode	: BYTE;
	wReadAddress	: WORD;
	wReadQuantity	: WORD;
	wWriteAddress	: WORD;
	wWriteQuantity	: WORD;
	//oStatus			: FbResult;
END_VAR
VAR
	index			: INT;
	xFound			: BOOL;
END_VAR
// Check to ensure the data model access was a succes
(*CASE oStatus.GetID() OF
	
	eErrorModbus.OK:
		
		// Assume NOT found
		xFound := FALSE;
		
		// Should add to some sort of data structure
		FOR index := 1 TO MAX_CONNECTIONS BY 1 DO
			IF ((m_ConnectionList[index].xActive) AND (m_ConnectionList[index].ipAddress = sClientId)) THEN

				// It exists
				xFound := TRUE;	
				
				// Update timer / counts
				//connectionList[index].xActive := TRUE;
				//connectionList[index].ipAddress := sClientId;
				m_ConnectionList[index].bUnitId := bUnitId;
				m_ConnectionList[index].bFunctionCode := bFunctionCode;
				m_ConnectionList[index].wReadAddress := wReadAddress;
				m_ConnectionList[index].uiReadQuantity := TO_UINT(wReadQuantity);
				m_ConnectionList[index].uiReadQuantityTotal := m_ConnectionList[index].uiReadQuantityTotal + TO_UINT(wReadQuantity);
				m_ConnectionList[index].wWriteAddress := wWriteAddress;
				m_ConnectionList[index].uiWriteQuantity := TO_UINT(wWriteQuantity);
				m_ConnectionList[index].uiWriteQuantityTotal := m_ConnectionList[index].uiWriteQuantityTotal + TO_UINT(wWriteQuantity);

				
				// Reset the timeout
				m_ConnectionList[index].commLossTimer(IN := FALSE, PT := stModbusServer.tTimeOut);
				
				// Exit the loop
				EXIT;
				
			END_IF
		END_FOR;
		
		IF (NOT xFound) THEN
			
			// Add to list
			FOR index := 1 TO MAX_CONNECTIONS BY 1 DO
				// Find first avilable spot in list
				IF (NOT m_ConnectionList[index].xActive) THEN

					// Add here
					m_ConnectionList[index].xActive := TRUE;
					m_ConnectionList[index].ipAddress := sClientId;
					m_ConnectionList[index].bUnitId := bUnitId;
					m_ConnectionList[index].bFunctionCode := 0;
					m_ConnectionList[index].wReadAddress := 0;
					m_ConnectionList[index].uiReadQuantity := 0;
					m_ConnectionList[index].uiReadQuantityTotal := 0;
					m_ConnectionList[index].wWriteAddress := 0;
					m_ConnectionList[index].uiWriteQuantity := 0;
					m_ConnectionList[index].uiWriteQuantityTotal := 0;
					m_ConnectionList[index].commLossTimer(IN := FALSE, PT := stModbusServer.tTimeOut);
					
					// Exit the loop
					EXIT;
				
				END_IF
			END_FOR;
		
		END_IF
		
ELSE

	// All other events - Do Nothing
	
	// eErrorModbus.INVALID_FRAME_LENGTH is the only other event I have encountered during testing.
	// This event was generated when a Wago PLC with a Master function block communicating had its
	// ethernet cable unplugged and plugged back in. <JAISON>

END_CASE
*)
END_METHOD

// NOT IMPLIMENTED FOR BECKHOFF AS IT DOES NOT SUPPORT THIS FUNCTIONALITY <JAISON>

(* ---------------------------------------------------------------------------
Func name   : 	beforeAccess
Description : 	Data access listener interface routine for the modbus server
				TCP connection which is called BEFORE any access to the modbus
				data model spaces.
Inputs      :	sClientId		-	IP Address of the connected client
				bUnitId			-	Unit id of the requested data model
				bFunctionCode	-	Modbus function code used to access data model
				wReadAddress	-	Address of data model read request
				wReadQuantity	-	Quantity of registers being read (in BOOL or WORD)
				wWriteAddress	-	Address of data model write request
				wWriteQuantity	-	Quantity of registers being written (in BOOL or WORD)
Returns     : 	USINT			-	Return 0 to allow data model access, any other return
									will deny access.
Notes       : 	
--------------------------------------------------------------------------- *)

METHOD beforeAccess : USINT
VAR_INPUT
	sClientId		: STRING(20);	// who is asking
	bUnitId			: BYTE;			// unit id of the requested data model
	bFunctionCode	: BYTE;
	wReadAddress	: WORD;
	wReadQuantity	: WORD;
	wWriteAddress	: WORD;
	wWriteQuantity	: WORD;
END_VAR
// This is where access to the data model can be monitored and prevented.
// If this function returns anything <> 0 access will be denyed. <JAISON>

beforeAccess := 0; // Return 0 to allow access to data model
END_METHOD

(* ---------------------------------------------------------------------------
Func name   : 	FB_exit
Description : 	Destructor
Inputs      :	None
Returns     : 	None
Notes       : 	
--------------------------------------------------------------------------- *)

METHOD FB_exit : BOOL
VAR_INPUT
	bInCopyCode : BOOL; // if TRUE, the exit method is called for exiting an instance that is copied afterwards (online change)
END_VAR
// Do nothing
END_METHOD

(* ---------------------------------------------------------------------------
Func name   : 	FB_init
Description : 	Constructor
Inputs      :	pDataAddessListener	:	pointer to function block which impliments
										the I_DataAccessListener interface.  If
										"_NULL" is passed in the server will use
										the internal listener.
Returns     : 	None
Notes       : 	
--------------------------------------------------------------------------- *)

METHOD FB_init : BOOL
VAR_INPUT
	bInitRetains 		: BOOL; // if TRUE, the retain variables are initialized (warm start / cold start)
    bInCopyCode  		: BOOL; // if TRUE, the instance afterwards gets moved into the copy code (online change)
	//pDataAddessListener	: POINTER TO I_DataAccessListener; // Set to "_NULL" to use built in server listener
END_VAR
VAR
	index			: INT;
END_VAR
//IF (pDataAddessListener <> _NULL) THEN

	// Register input function block to listen for any server requests
	//m_ModbusSlave.RegisterDataAccessListener(I_DataAccessListener:= pDataAddessListener^);

//ELSE

	// Register this function block to listen for any server requests
	//m_ModbusSlave.RegisterDataAccessListener(I_DataAccessListener:= THIS^);

//END_IF

// Inialize the connection list
FOR index := 1 TO MAX_CONNECTIONS BY 1 DO
		
	m_ConnectionList[index].xActive := FALSE;
	m_ConnectionList[index].ipAddress := 'INACTIVE';
	m_ConnectionList[index].bUnitId := 0;
	m_ConnectionList[index].bFunctionCode := 0;
	m_ConnectionList[index].wReadAddress := 0;
	m_ConnectionList[index].uiReadQuantity := 0;
	m_ConnectionList[index].uiReadQuantityTotal := 0;
	m_ConnectionList[index].wWriteAddress := 0;
	m_ConnectionList[index].uiWriteQuantity := 0;
	m_ConnectionList[index].uiWriteQuantityTotal := 0;
	m_ConnectionList[index].commLossTimer(IN := FALSE, PT := stModbusServer.tTimeOut);
	
END_FOR
END_METHOD

(* ---------------------------------------------------------------------------
Func name   : 	GetCoilPointer
Description : 	Returns a pointer to the BOOL Coils array.
Inputs      :	None
Returns     : 	POINTER TO BOOL	-	Pointer to the Coils BOOL array.
Notes       : 	Use this method as an input to a memcopy routine with any
				required offset in order to overlay the data onto a more
				useful BOOL aligned struct. 
--------------------------------------------------------------------------- *)

METHOD GetCoilPointer : POINTER TO BOOL
VAR_INPUT
END_VAR
GetCoilPointer := ADR(gaxCoils);
END_METHOD

(* ---------------------------------------------------------------------------
Func name   : 	GetDiscreteInputPointer
Description : 	Returns a pointer to the BOOL Discrete Inputs array.
Inputs      :	None
Returns     : 	POINTER TO BOOL	-	Pointer to the Discrete Inputs BOOL array.
Notes       : 	Use this method as an input to a memcopy routine with any
				required offset in order to overlay the data onto a more
				useful BOOL aligned struct. 
--------------------------------------------------------------------------- *)

METHOD GetDiscreteInputPointer : POINTER TO BOOL
VAR_INPUT
END_VAR
GetDiscreteInputPointer := ADR(gaxDiscreteInputs);
END_METHOD

(* ---------------------------------------------------------------------------
Func name   : 	GetHoldingRegisterPointer
Description : 	Returns a pointer to the WORD Holding Registers array.
Inputs      :	None
Returns     : 	POINTER TO WORD	-	Pointer to the Holding Resgisters WORD array.
Notes       : 	Use this method as an input to a memcopy routine with any
				required offset in order to overlay the data onto a more
				useful WORD aligned struct. 
--------------------------------------------------------------------------- *)

METHOD GetHoldingRegisterPointer : POINTER TO WORD
VAR_INPUT
END_VAR
GetHoldingRegisterPointer := ADR(gawHoldingRegisters);
END_METHOD

(* ---------------------------------------------------------------------------
Func name   : 	GetInputRegisterPointer
Description : 	Returns a pointer to the WORD Input Registers array.
Inputs      :	None
Returns     : 	POINTER TO WORD	-	Pointer to the Input Resgisters WORD array.
Notes       : 	Use this method as an input to a memcopy routine with any
				required offset in order to overlay the data onto a more
				useful WORD aligned struct. 
--------------------------------------------------------------------------- *)

METHOD GetInputRegisterPointer : POINTER TO WORD
VAR_INPUT
END_VAR
GetInputRegisterPointer := ADR(gawInputRegisters);
END_METHOD

// NOT IMPLIMENTED FOR BECKHOFF AS IT DOES NOT SUPPORT THIS FUNCTIONALITY <JAISON>

(* ---------------------------------------------------------------------------
Func name   : 	IsClientConnected
Description : 	Check for the connection status of a specific client,
				defined by its IP Address.
				to the server and FALSE if not.
Inputs      :	sClientId	-	IP Address of the client to check
Returns     : 	BOOL		-	TRUE if connected, otherwise FALSE
Notes       : 	Use this method to cyclically poll the server for a specific 
				client's connection status.
--------------------------------------------------------------------------- *)

METHOD IsClientConnected : BOOL
VAR_INPUT
	sClientId		: STRING(20);
END_VAR
VAR
	index			: INT;
	xFound			: BOOL;
END_VAR
// Assume station doesnt exist
(*xFound := FALSE;

// Should add to some sort of data structure
FOR index := 1 TO MAX_CONNECTIONS BY 1 DO
	IF ((m_ConnectionList[index].xActive) AND (m_ConnectionList[index].ipAddress = sClientId)) THEN

		// It exists
		xFound := TRUE;
				
		// Exit the loop
		EXIT;
				
	END_IF
END_FOR;

IsClientConnected := xFound;*)
END_METHOD

// NOT IMPLIMENTED FOR BECKHOFF AS IT DOES NOT SUPPORT THIS FUNCTIONALITY <JAISON>

(* ---------------------------------------------------------------------------
Func name   : 	UpdateConnectionList
Description : 	Private method used to encapsulate the connection list
				update logic.
Inputs      :	None
Returns     : 	UINT		-	Number of connected clients to the server
Notes       : 	This method needs to be run every scan to properly updated
				the connection list and refresh the number of connected
				clients.
--------------------------------------------------------------------------- *)

METHOD PRIVATE UpdateConnectionList : UINT
VAR_INPUT
END_VAR
VAR
	index			: INT;
	numConnected	: UINT;
END_VAR
// Assume no connections
(*numConnected := 0;

// Should add to some sort of data structure
FOR index := 1 TO MAX_CONNECTIONS BY 1 DO

	// Check if connection is actve
	IF (m_ConnectionList[index].xActive) THEN
		
		// Increase the number of connections
		numConnected := numConnected + 1;
	
		// Run the timeout timer
		m_ConnectionList[index].commLossTimer(IN:= TRUE);
	
		// Check for timeout
		IF (m_ConnectionList[index].commLossTimer.Q) THEN
			
			// Decrease the number of connections
			numConnected := numConnected - 1;
		
			// Remove from connection list
			m_ConnectionList[index].xActive := FALSE;
			m_ConnectionList[index].ipAddress := 'INACTIVE';
			m_ConnectionList[index].bUnitId := 0;
			m_ConnectionList[index].bFunctionCode := 0;
			m_ConnectionList[index].wReadAddress := 0;
			m_ConnectionList[index].uiReadQuantity := 0;
			m_ConnectionList[index].uiReadQuantityTotal := 0;
			m_ConnectionList[index].wWriteAddress := 0;
			m_ConnectionList[index].uiWriteQuantity := 0;
			m_ConnectionList[index].uiWriteQuantityTotal := 0;
			m_ConnectionList[index].commLossTimer(IN := FALSE, PT := stModbusServer.tTimeOut);
		
		END_IF
	
	END_IF
	
END_FOR

// return connection count
UpdateConnectionList := numConnected;
*)
END_METHOD

END_FUNCTION_BLOCK

// 20 Program Organization Units/Modbus/fb_ReadHoldingRegisters
(*AUTHOR:			Jaison Schaab*)
(*DATE:				March 4 / 2021*)
(*DESCRIPTION: 		This Function Block will perform a Modbus Master FC03 Read of Holding Registers*)

(*NOTES:
*
*	The Beckhoff documentation talks about "Output" registers which are actually 'Holding" registers which can be read or written to.
*	By passing in a TRUE to the "xRead" input the block will read as fast as it can usually taking 3 PLC scans per read, if you want
* 	this to run slower you can connect a timed trigger to the "xRead" input to trigger the read when desired.
*	<TEST>
*	Through empirical testing I have found that the Beckhoff master write will only handle data chunks of 125 WORDS (250 BYTES) MAX.  So multiple 
*	master requests will be required to handle larger data transfers. <JAISON>
*
*	If the requested "uiLength" is too large (ie. over the limit mentioned above) the "nErrId" will return the code 32771. 
*
*)

(*UPDATE: 			March. 18 2021 - Jaison Schaab

					Code Ported from Wago.
					
					Code Is fully tested and functional.
*)

FUNCTION_BLOCK fb_ReadHoldingRegisters
VAR_INPUT
	xEnable					: BOOL;						// Input to enable the Block
	xRead					: BOOL;						// Single cycle pulse to start read (Will be ignored if Modbus Master is busy)
	uiLength				: UINT;						// Length of the data to be read in BYTES. MUST BE LESS THAN 125 WORDS or 250 BYTES.  Based on Empirical testing. <JAISON>
	pDataAddr				: POINTER TO WORD;			// Pointer to data space where read data will be copied to
	uiMBAddr 				: UINT;						// Modbus address where data resides on the server			
	stModbusTarget 			: TModbusTargetConfig ;		// Modbus Target object containing information on the server
END_VAR	
VAR_OUTPUT
	xUpdate					: BOOL;						// Output when TRUE symbolizes data has been read and is ready for program to update
	xComFailure				: BOOL;						// Output when TRUE symbolizes modbus communication failure
END_VAR
VAR
	// Modbus Comm Block Status
	xBusy					: BOOL;						// TRUE when Modbus Master block is busy
	xError					: BOOL;						// TRUE when Modbus function block error occurs
	nErrId					: UDINT;					// ADS error number when xError is SET
	uiQuantityRead			: UDINT;					// Contains the number of bytes read
	
	// Modbus Comm Control Variables			
	ReadDoneTrigger			: F_TRIG;					// Falling edge trigger to signify the Read completion
		
	fbMBReadRegs			: FB_MBReadRegs;			// Modbus Read Holding Registers (Function Code 3)
	
	fbModbusError			: fb_ModbusError;			// Modbus communication error check
END_VAR
VAR CONSTANT
	//tConnectionResetTimeout	: TIME := T#5S;				// Connection Reset delay timeout
END_VAR

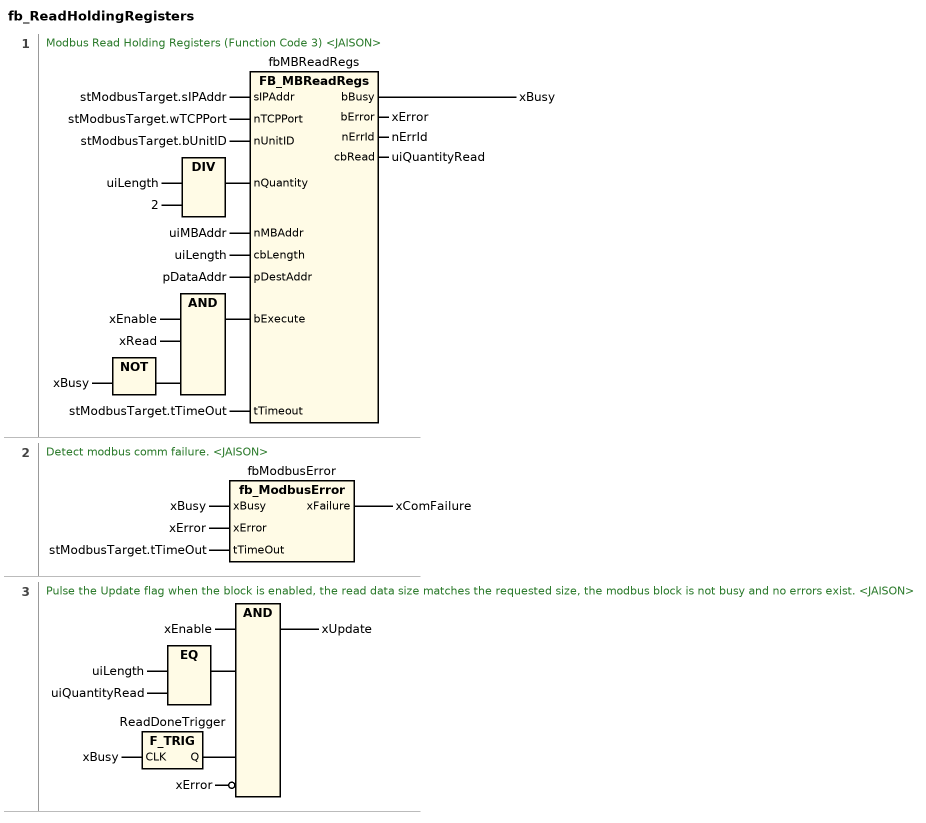
// NETWORK 1
// Modbus Read Holding Registers (Function Code 3) <JAISON>
fbMBReadRegs(
    sIPAddr := stModbusTarget.sIPAddr,
    nTCPPort := stModbusTarget.wTCPPort,
    nUnitID := stModbusTarget.bUnitID,
    nQuantity := uiLength / 2,
    nMBAddr := uiMBAddr,
    cbLength := uiLength,
    pDestAddr := pDataAddr,
    bExecute := xEnable AND xRead AND NOT xBusy,
    tTimeout := stModbusTarget.tTimeOut,
    bError => xError,
    nErrId => nErrId,
    cbRead => uiQuantityRead); // FB_MBReadRegs
xBusy := fbMBReadRegs.bBusy;

// NETWORK 2
// Detect modbus comm failure. <JAISON>
fbModbusError(xBusy := xBusy, xError := xError, tTimeOut := stModbusTarget.tTimeOut); // fb_ModbusError
xComFailure := fbModbusError.xFailure;

// NETWORK 3
// Pulse the Update flag when the block is enabled, the read data size matches the requested size, the modbus block is not busy and no errors exist. <JAISON>
ReadDoneTrigger(CLK := xBusy); // F_TRIG
xUpdate := xEnable AND uiLength = uiQuantityRead AND ReadDoneTrigger.Q AND NOT xError;

END_FUNCTION_BLOCK

// 20 Program Organization Units/Modbus/fb_ReadInputRegisters
(*AUTHOR:			Jaison Schaab*)
(*DATE:				March 4 / 2021*)
(*DESCRIPTION: 		This Function Block will perform a Modbus Master FC04 Read of Input Registers*)

(*NOTES:
*
*	By passing in a TRUE to the "xRead" input the block will read as fast as it can usually taking 3 PLC scans per read, if you want
* 	this to run slower you can connect a timed trigger to the "xRead" input to trigger the read when desired.
*
*	Through empirical testing I have found that the Beckhoff master read will only handle data chunks of 125 WORDS (250 BYTES) MAX.  So multiple 
*	master requests will be required to handle larger data transfers. <JAISON>
*
*	If the requested "uiLength" is too large (ie. over the limit mentioned above) the "nErrId" will return the code 32771. 
*
*)

(*UPDATE: 			March. 18 2021 - Jaison Schaab

					Code Ported from Wago.
					
					Code Is fully tested and functional.
*)

FUNCTION_BLOCK fb_ReadInputRegisters
VAR_INPUT
	xEnable					: BOOL;						// Input to enable the Block
	xRead					: BOOL;						// Single cycle pulse to start read (Will be ignored if Modbus Master is busy)
	uiLength				: UINT;						// Length of the data to be read in BYTES. MUST BE LESS THAN 125 WORDS or 250 BYTES.  Based on Empirical testing. <JAISON>
	pDataAddr				: POINTER TO WORD;			// Pointer to data space where read data will be copied to
	uiMBAddr 				: UINT;						// Modbus address where data resides on the server			
	stModbusTarget 			: TModbusTargetConfig ;		// Modbus Target object containing information on the server
END_VAR	
VAR_OUTPUT
	xUpdate					: BOOL;						// Output when TRUE symbolizes data has been read and is ready for program to update
	xComFailure				: BOOL;						// Output when TRUE symbolizes modbus communication failure
END_VAR
VAR
	// Modbus Comm Block Status
	xBusy					: BOOL;						// TRUE when Modbus Master block is busy
	xError					: BOOL;						// TRUE when Modbus Master function block error occurs
	nErrId					: UDINT;					// ADS error number when xError is SET
	uiQuantityRead			: UDINT;					// Contains the number of bytes read
	
	// Modbus Comm Control Variables	
	ReadDoneTrigger			: F_TRIG;					// Falling edge trigger to signify the Read completion

	fbMBReadInputRegs		: FB_MBReadInputRegs;		// Modbus Read Input Registers (Function Code 4)
		
	fbModbusError			: fb_ModbusError;			// Modbus communication error check
END_VAR

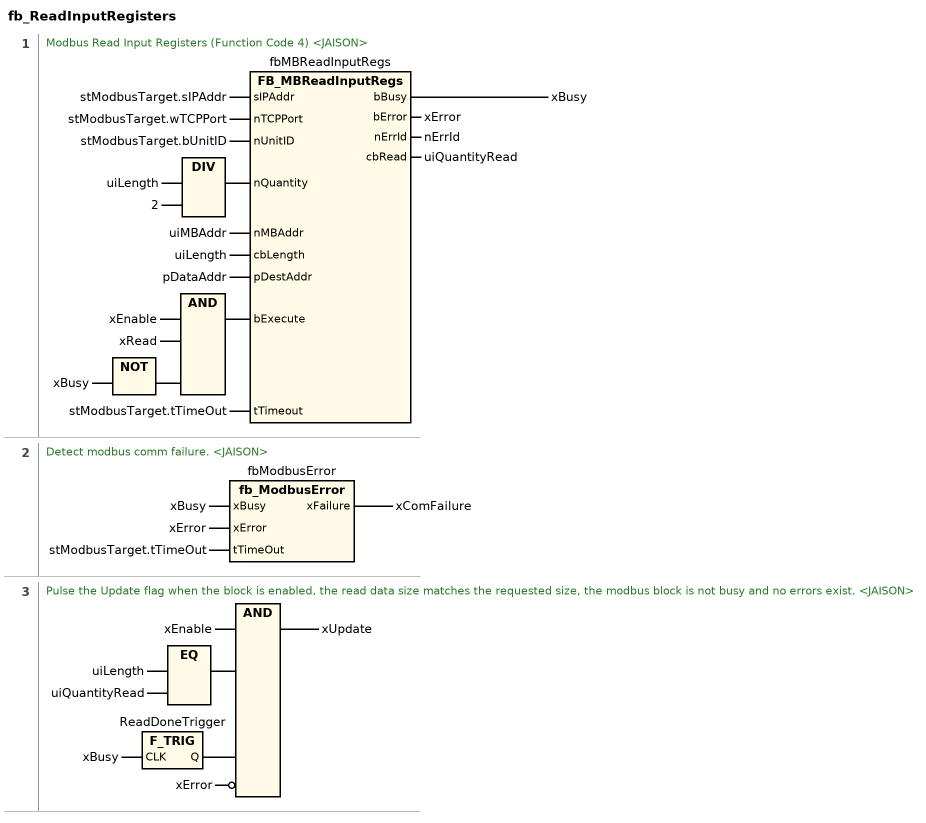
// NETWORK 1
// Modbus Read Input Registers (Function Code 4) <JAISON>
fbMBReadInputRegs(
    sIPAddr := stModbusTarget.sIPAddr,
    nTCPPort := stModbusTarget.wTCPPort,
    nUnitID := stModbusTarget.bUnitID,
    nQuantity := uiLength / 2,
    nMBAddr := uiMBAddr,
    cbLength := uiLength,
    pDestAddr := pDataAddr,
    bExecute := xEnable AND xRead AND NOT xBusy,
    tTimeout := stModbusTarget.tTimeOut,
    bError => xError,
    nErrId => nErrId,
    cbRead => uiQuantityRead); // FB_MBReadInputRegs
xBusy := fbMBReadInputRegs.bBusy;

// NETWORK 2
// Detect modbus comm failure. <JAISON>
fbModbusError(xBusy := xBusy, xError := xError, tTimeOut := stModbusTarget.tTimeOut); // fb_ModbusError
xComFailure := fbModbusError.xFailure;

// NETWORK 3
// Pulse the Update flag when the block is enabled, the read data size matches the requested size, the modbus block is not busy and no errors exist. <JAISON>
ReadDoneTrigger(CLK := xBusy); // F_TRIG
xUpdate := xEnable AND uiLength = uiQuantityRead AND ReadDoneTrigger.Q AND NOT xError;

END_FUNCTION_BLOCK

// 20 Program Organization Units/Modbus/fb_WriteHoldingRegisters
(*AUTHOR:			Jaison Schaab*)
(*DATE:				March 4 / 2021*)
(*DESCRIPTION: 		This Function Block will perform a Modbus Master FC16 Write of Holding Registers*)

(*NOTES:
*
*	The Beckhoff documentation talks about "Output" registers which are actually 'Holding" registers which can be read or written to.
*	By passing in a TRUE to the "xWrite" input the block will write as fast as it can usually taking 3 PLC scans per write, if you want
* 	this to run slower you can connect a timed trigger to the "xWrite" input to trigger the write when desired.
*
*	Through empirical testing I have found that the Beckhoff master write will only handle data chunks of 123 WORDS (246 BYTES) MAX.  So multiple 
*	master requests will be required to handle larger data transfers. <JAISON>
*
*	If the requested "uiLength" is too large (ie. over the limit mentioned above) the "nErrId" will return the code 32771. 
*
*)

(*UPDATE: 			March. 18 2021 - Jaison Schaab

					Code Ported from Wago.
					
					Code Is fully tested and functional.
*)

FUNCTION_BLOCK fb_WriteHoldingRegisters
VAR_INPUT
	xEnable					: BOOL;						// Input to enable the Block
	xWrite					: BOOL;						// Single cycle pulse to start write (Will be ignored if Modbus Master is busy)
	uiLength				: UINT;						// Length of the data to be written in BYTES. MUST BE LESS THAN 123 WORDS or 246 BYTES. Based on Empirical testing. <JAISON>
	pDataAddr				: POINTER TO WORD;			// Pointer to data space where written data will be copied from
	uiMBAddr 				: UINT;						// Modbus address where data resides on the server		
	stModbusTarget 			: TModbusTargetConfig ;		// Modbus Target object containing information on the server
END_VAR
VAR_OUTPUT
	xReady					: BOOL;						// Output when TRUE symbolizes data has been written and is ready for another write
	xComFailure				: BOOL;						// Output when TRUE symbolizes modbus communication failure
END_VAR
VAR
	// Modbus Comm Block Status
	xBusy					: BOOL;						// TRUE when Modbus Master block is busy
	xError					: BOOL;						// TRUE when Modbus Master function block error occurs
	nErrId					: UDINT;					// ADS error number when xError is SET
	uiQuantityWrote			: UDINT;					// Contains the number of bytes written
	
	// Modbus Comm Control Variables
	WriteDoneTrigger		: F_TRIG;					// Falling edge trigger to signify the Write completion
	DataReadyBistable		: RS;						// Data write ready bi-stable

	fbMBWriteRegs			: FB_MBWriteRegs;			// Modbus Write Holding Registers (Function Code 16)
	
	fbModbusError			: fb_ModbusError;			// Modbus communication error check
END_VAR

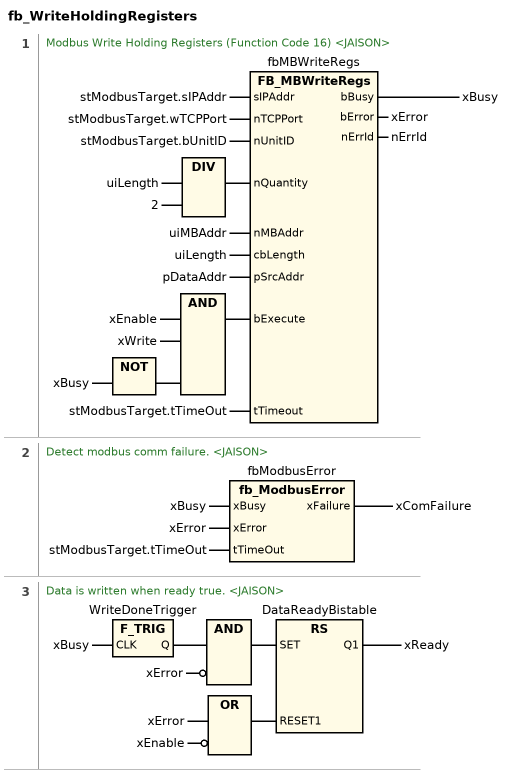
// NETWORK 1
// Modbus Write Holding Registers (Function Code 16) <JAISON>
fbMBWriteRegs(
    sIPAddr := stModbusTarget.sIPAddr,
    nTCPPort := stModbusTarget.wTCPPort,
    nUnitID := stModbusTarget.bUnitID,
    nQuantity := uiLength / 2,
    nMBAddr := uiMBAddr,
    cbLength := uiLength,
    pSrcAddr := pDataAddr,
    bExecute := xEnable AND xWrite AND NOT xBusy,
    tTimeout := stModbusTarget.tTimeOut,
    bError => xError,
    nErrId => nErrId); // FB_MBWriteRegs
xBusy := fbMBWriteRegs.bBusy;

// NETWORK 2
// Detect modbus comm failure. <JAISON>
fbModbusError(xBusy := xBusy, xError := xError, tTimeOut := stModbusTarget.tTimeOut); // fb_ModbusError
xComFailure := fbModbusError.xFailure;

// NETWORK 3
// Data is written when ready true. <JAISON>
WriteDoneTrigger(CLK := xBusy); // F_TRIG
DataReadyBistable(SET := WriteDoneTrigger.Q AND NOT xError, RESET1 := xError OR NOT xEnable); // RS
xReady := DataReadyBistable.Q1;

END_FUNCTION_BLOCK

// 20 Program Organization Units/Process Calculation Functions/f_CalculateDensityPPAfromSGU
(* ---------------------------------------------------------------------------
Func name   : 	f_CalculateDensityPPAfromSGU
Description : 	Function to calculate and return the density lbs per proppant added [PPA].
				
Inputs      :	baseDensity	in [SGU]
				proppantDensity	in [SGU]
				measuredDensity in [SGU]

Returns     : 	REAL	-	The density value in density unit [PPA]
Notes       : 	
--------------------------------------------------------------------------- *)

(*UPDATE: 			March. 18 2021 - Jaison Schaab

					Code Ported from Wago.
					
					Code has NOT Yet been tested.
*)

FUNCTION f_CalculateDensityPPAfromSGU : REAL
VAR_INPUT
	baseDensity		: REAL;			// base density [SGU]
	proppantDensity	: REAL;			// proppant density [SGU]
	measuredDensity	: REAL;			// measured density [SGU]
END_VAR
VAR
END_VAR
VAR CONSTANT
	CONVERSION_FACTOR	: REAL := 8.345;				// conversion factor [SGU] to [PPG]
END_VAR

(*
														Mixture Density	-	Base Density
			PPA				=		8.345			x	_________________________________
																 Mixture Density
														1	-	_________________
																Proppant Density
															
															
															
																[SGU] 		- 		[SGU]		
		[lbs / proppant added]	=	 Conversion Factor	x	_________________________________
																		  [SGU]
															1	-	__________________
																		  [SGU]
*)


f_CalculateDensityPPAfromSGU	:=	CONVERSION_FACTOR	* ( measuredDensity - baseDensity )	/	( 1.0 - (measuredDensity / proppantDensity ) );

END_FUNCTION

// 20 Program Organization Units/Process Calculation Functions/f_CalculateDensityPPGfromSGU
(* ---------------------------------------------------------------------------
Func name   : 	f_CalculateDensityPPGfromSGU
Description : 	Function to calculate and return the density PPG
				in unit of [lbs/gal]. Conversion factor of 8.345.
Inputs      :	measuredDensity	in [SGU]
Returns     : 	REAL	-	The density value in density unit PPG [lbs/gal]
Notes       : 	
--------------------------------------------------------------------------- *)

(*UPDATE: 			March. 18 2021 - Jaison Schaab

					Code Ported from Wago.
					
					Code has NOT Yet been tested.
*)

FUNCTION f_CalculateDensityPPGfromSGU : REAL
VAR_INPUT
	measuredDensity		: REAL;				// measured density [SGU]
END_VAR
VAR
END_VAR
VAR CONSTANT
	CONVERSION_FACTOR	: REAL := 8.345;	// conversion factor [SGU] to [PPG]
END_VAR

(*
 		PPG Density				=	Conversion Factor  	x 	Corrected Density
		
		[lbs/gal]				=		8.345			x		[SGU]
*)

f_CalculateDensityPPGfromSGU	:= CONVERSION_FACTOR 	* 	measuredDensity;

END_FUNCTION

// 20 Program Organization Units/Testing Functions/FB_CNTRLSYS_RESPONSE
(*AUTHOR:		Graham Hunter*)
(*DATE:			November 11, 2020 *)
(*DESCRIPTION:	This function block determines the fundamental Control System response by determining the peak or valley values & times as well as settling value & time
				for a step change in the Plant Dynamics. To test the Peak, Valley, or Settling system response, set the m_TestPeak, m_TestValley, or m_TestSettlingTime variables true on a step change.
*)
(*NOTES:		*)	
	
FUNCTION_BLOCK FB_CNTRLSYS_RESPONSE
VAR_INPUT
	uiCycleTime_us				: UINT; // scan cycle time [us]
	xEnable						: BOOL; // Enable this function block	
	m_CurrentSP					: REAL; // Current Set-point [%]
	m_OldFeedback				: REAL; // Old feedback value in scan cycle (farthest from where this fb is called)	[%]					
	m_NewFeedback				: REAL; // New feedback value in scan cycle (closest to where this fb is called) [%]
END_VAR
VAR_OUTPUT
	m_PeakTime					: TIME; // Final Peak time [s]
	m_ValleyTime				: TIME; // Final Valley time [s]
	m_SettlingTime				: TIME; // Final Settling time [s]
	m_LastMaxValue				: REAL; // Final Peak Value [%]
	m_LastMinValue				: REAL;	// Final Valley Value [%]
END_VAR
VAR_IN_OUT
	m_TestPeak					: BOOL; // Start Peak Test
	m_TestValley				: BOOL; // Start Valley Test
	m_TestSettlingTime			: BOOL; // Start Settling Time Test
END_VAR
VAR
	// Timers
	m_TestPeakTON				: TON; 				// peak timer
	m_TestValleyTON				: TON;				// valley timer
	m_TestSettlingTON			: TON;				// settling timer
	m_ValueRunningAverage		: FB_RUNNING_AVG;	// Running average of feedback value (not used currently)
	m_FirstPeak					: BOOL;				// indication of first peak reached
	m_FirstValley				: BOOL;				// indication of first valley reached
	m_FirstSettlingTime			: BOOL;				// indication of settling time reached (error within 2% of setpoint)
END_VAR

IF xEnable THEN
	
	IF m_TestPeak THEN
		IF (m_NewFeedback > m_OldFeedback) AND NOT m_FirstPeak THEN
			m_TestPeakTON(IN := TRUE, PT := T#20000S);
			m_LastMaxValue := m_NewFeedback;
			m_PeakTime 	   := m_TestPeakTON.ET;
		// ELSE
			// m_TestPeakTON(IN := FALSE);
		ELSIF m_NewFeedback < m_OldFeedback THEN
			m_FirstPeak := TRUE;
			m_TestPeak := FALSE;
			m_TestPeakTON(IN := FALSE);
		END_IF
	ELSE
		m_FirstPeak := FALSE;
	END_IF
	
	IF m_TestValley THEN
		IF (m_NewFeedback < m_OldFeedback) AND NOT m_FirstValley THEN
			m_TestValleyTON(IN := TRUE, PT := T#20000S);
			m_LastMinValue := m_NewFeedback;
			m_ValleyTime :=  	m_TestValleyTON.ET;
		// ELSE
			// m_TestValleyTON(IN := FALSE);	
		ELSIF m_NewFeedback > m_OldFeedback THEN
			m_FirstValley:= TRUE;
			m_TestValley := FALSE;
			m_TestValleyTON(IN := FALSE);
		END_IF
	ELSE
		m_FirstValley := FALSE;
	END_IF
	
	IF m_TestSettlingTime THEN
		m_TestSettlingTON(IN := TRUE, PT := T#20000S);
		//m_TestSettlingTON.ET;
		IF ABS(m_CurrentSP - m_NewFeedback) > 2.0 THEN
			m_SettlingTime :=  	m_TestSettlingTON.ET;
		ELSE 
			;
		END_IF
	ELSE
		m_TestSettlingTON(IN := FALSE);
	END_IF

ELSE
	;
END_IF

END_FUNCTION_BLOCK

// 20 Program Organization Units/Utility Functions/Statistic Functions/FB_RUNNING_AVG
(*AUTHOR:		Port over from C++ library*)
(*DATE:			 *)
(*DESCRIPTION:	This Function takes in an rINPUT data point value with an overall N buffer number of data points and outputs an average value of rINPUT.*)

(*NOTES:		*)

FUNCTION_BLOCK FB_RUNNING_AVG
VAR_INPUT
	rINPUT		: REAL;
	N			: INT;
END_VAR
VAR_OUTPUT
	rAVG_OUPUT	: REAL;
END_VAR
VAR
	
	rValues: ARRAY[0..20000] OF REAL;	// This buffer contains the values to be averaged 
	iCounter	: INT;
	rSum		: REAL;
	i			: INT;
END_VAR

IF N <= 1 THEN
    N := 1;
END_IF
(* Start loading the array with values *)
IF iCounter >= N THEN
    iCounter := 0;
ELSIF iCounter < 0 THEN
    iCounter := 0;
END_IF
//remove old average from the sum
rSum := rSum - rValues[iCounter];
rSum := rSum + rInput;
rValues[iCounter] := rInput;
rAVG_OUPUT := rSum / N;
(* increment the counter for loading the array *)
iCounter := iCounter + 1;

END_FUNCTION_BLOCK

// 20 Program Organization Units/Testing Functions/fb_TriStateValveSimulator
(*AUTHOR:			Jaison Schaab*)
(*DATE:				March. 9 / 2020*)
(*DESCRIPTION: 		Simulation for a Tri-State valve which is controlled by
					a digitial (BOOL) open/close actuator signal.  This block
					will provide both digital (BOOL) open/close and analog
					valve position feedback signals which are based on a
					configurable input delay time*)

(*NOTES:			The Open value can be smaller, larger or equal to the Close value.
					The logic will automatically decode the valve state in any scaling
					situaltion.
*)					

(*UPDATE: 			March. 18 2021 - Jaison Schaab

					Code Ported from Wago.
					
					Code has NOT Yet been tested.
*)

(*UPDATE: 			September. 1 2020 - Jaison Schaab

					Changed the Opened/Closed bi-stable feeback blocks to ONLY shift when the opposite
					output is given and NOT when the actuator output is removed.  This is because  on the 
					E-Frac dual-action valve the outputs are disabled even when the valve remains closed/opened.
*)			

FUNCTION_BLOCK fb_TriStateValveSimulator
VAR_INPUT
	xOpenActuator		: BOOL;					// Open actuator input from the valve control block
	xCloseActuator		: BOOL;					// Close actuator input from the valve control block
	tValveShiftingDelay	: TIME;					// Amount of time simulated valve will take to shift
	rOpenValue			: REAL;					// Valve opened feedback value (used for scaling rValvePosition output)
	rCloseValue			: REAL;					// Valve closed feedback value (used for scaling rValvePosition output)
	uiCycleTime_us		: UINT;					// PLC cycle time in Microseconds (us)
END_VAR
VAR_OUTPUT
	xOpenedFeedback		: BOOL;					// Opened feedback output for valve control block
	xClosedFeedback		: BOOL;					// Closed feedback output for valve control block
	rValvePosition		: REAL;					// Analog valve position feedback for valve control block
END_VAR
VAR
	OpenDelayTimer		: TON;					// Timer for valve open delay
	CloseDelayTimer		: TON;					// Timer for valve close delay
	
	OpenBiStable		: RS;					// Triggers for valve open digital feedback
	CloseBiStable		: RS;					// Triggers for valve close digital feedback
	
	rValveShiftSlice	: REAL;					// Amount the simulated analog valve position shifts per PLC cycle
	
	lrSecondsCycleTime	: LREAL;				// PLC cycle time in seconds (s)
	lrNumShiftSlices	: LREAL;				// Number of PLC cycles required to fully shift the valve, based on the input shift delay time
	lrShiftDelaySeconds	: LREAL;				// Simulated valve shift delay in seconds (S), based on the input shift delay time
END_VAR
VAR CONSTANT
	 US_TO_SECONDS_MULT : LREAL := 0.000001;	// microseconds (us) to seconds multiplier
	 MS_TO_SECONDS_MULT	: LREAL := 0.001;		// milliseconds (ms) to seconds multiplier
END_VAR

(* Open Valve Digital Feedback Simulation Logic *)

// Simulate Opened Feedback <JAISON>
// SET after Open shifting delay has expred
// RESET when valve Close is activated (ie. Open FALSE and Close TRUE)
//OpenBiStable(SET:= OpenDelayTimer.Q, RESET1:= ((NOT xOpenActuator) AND xCloseActuator), Q1=> xOpenedFeedback);
OpenBiStable(SET:= OpenDelayTimer.Q, RESET1:= xCloseActuator, Q1=> xOpenedFeedback);

// Simulate valve opening when actuators are properly set (ie. Close FALSE and Open TRUE) <JAISON>
OpenDelayTimer(IN:= ((NOT xCloseActuator) AND xOpenActuator), PT:= tValveShiftingDelay);

(* Close Valve Digital Feedback Simulation Logic *)

// Simulate Closed Feedback <JAISON>
// SET after Close shifting delay has expred
// RESET when valve Open is activated (ie. Close FALSE and Open TRUE)
//CloseBiStable(SET:= CloseDelayTimer.Q, RESET1:= ((NOT xCloseActuator) AND xOpenActuator), Q1=> xClosedFeedback);
CloseBiStable(SET:= CloseDelayTimer.Q, RESET1:= xOpenActuator, Q1=> xClosedFeedback);

// Simulate valve opening when actuators are properly set (ie. Open FALSE and Close TRUE) <JAISON>
CloseDelayTimer(IN:= ((NOT xOpenActuator) AND xCloseActuator), PT:= tValveShiftingDelay);

(* Analog Valve Position Simulation Logic *)

// Calculate the PLC cycle time (Slice) in seconds
// Ensure not to divide by 0
IF (uiCycleTime_us > 0) THEN
	lrSecondsCycleTime := TO_LREAL(uiCycleTime_us) * US_TO_SECONDS_MULT;
ELSE
	lrSecondsCycleTime := 1;
END_IF

// Calculate the valve shift time in seconds
lrShiftDelaySeconds := TIME_TO_LREAL(tValveShiftingDelay) * MS_TO_SECONDS_MULT;

// Calculate the number of PLC slices per valve shift
lrNumShiftSlices := lrShiftDelaySeconds / lrSecondsCycleTime;

// Calculate the amount of valve shift per PLC slice
IF (lrNumShiftSlices > 0) THEN
	rValveShiftSlice := TO_REAL(TO_LREAL(ABS(rCloseValue - rOpenValue)) / lrNumShiftSlices);
ELSE
	rValveShiftSlice := 1;
END_IF

//Simulate the valve position
IF (rCloseValue >= rOpenValue) THEN // CLOSE >= OPEN
	// Update valve position when opening
	IF (OpenDelayTimer.IN) THEN
		rValvePosition := MAX(rOpenValue, rValvePosition-rValveShiftSlice);
	END_IF

	// Updated valve position when closing
	IF (CloseDelayTimer.IN) THEN
		rValvePosition := MIN(rCloseValue, rValvePosition+rValveShiftSlice);
	END_IF
ELSE // CLOSE < OPEN
	// Update valve position when opening
	IF (OpenDelayTimer.IN) THEN
		rValvePosition := MIN(rOpenValue, rValvePosition+rValveShiftSlice);
	END_IF

	// Updated valve position when closing
	IF (CloseDelayTimer.IN) THEN
		rValvePosition := MAX(rCloseValue, rValvePosition-rValveShiftSlice);
	END_IF
END_IF

END_FUNCTION_BLOCK

// 20 Program Organization Units/Utility Functions/Conversion Functions/F_SPLIT_REGISTERS
(*AUTHOR:		James Belcher*)
(*DATE:			 *)
(*DESCRIPTION:	This Function handle resolution and 32 bits value by splitting most
				significant word and least significant word, and handles  *)

(*NOTES:		*)
		
FUNCTION F_SPLIT_REGISTERS : WORD
VAR_INPUT
	fInput: REAL;
	qIsMSB: BOOL;
	fGain: REAL;
	wOffset: WORD;
END_VAR
VAR
	dInput: DWORD;
	wLSB: WORD;
	wMSB: WORD;
END_VAR

dInput := REAL_TO_DWORD( ( fInput + wOffset ) * fGain );

// Splits most significant word and least significant word
wMSB := DWORD_TO_WORD( SHR( dInput , 16 ) * BOOL_TO_BYTE( qIsMSB ) );
wLSB := DWORD_TO_WORD( ( dInput AND 16#FFFF ) * BOOL_TO_BYTE( NOT qIsMSB ) );

// Outputs value of most or least significant word
F_SPLIT_REGISTERS := wMSB + wLSB;

///// RESOLUTION EXAMPLES /////
// 	fInput	:=  500.15
//	fGain	:= 10
// 	fOffset	:= 0

// dInput	:= ( 500.15 + 0 ) *  10
// dInput	:= 5001

// dInput	:= 5001
// fOutput	:= 5001 / 10 - 0 := 500.1

// 	fInput	:=  -25.5
//	fGain	:= 10
// 	fOffset	:= 50

// dInput	:= ( -25.5 + 50 ) *  10
// dInput	:= 30.5 * 10
// dInput	:= 305

///// 32BIT VALUE EXAMPLES /////
// DWORD := 123456789
// IR[0]	:= F_SPLIT_REGISTERS( DWORD , TRUE , 1 , 0 )		:= 1883
// IR[1]	:= F_SPLIT_REGISTERS( DWORD , FALSE , 1 , 0 )		:= 52501

END_FUNCTION

// 20 Program Organization Units/Utility Functions/Conversion Functions/F_STATUS_WORD_TO_WORD
(*AUTHOR:		James Belcher*)
(*DATE:			June 30, 2020 *)
(*DESCRIPTION:	This Function is to handle Status Word block conversion into Word *)

(*NOTES:		*)		
FUNCTION F_STATUS_WORD_TO_WORD : WORD
VAR_INPUT
	pBitPointer: POINTER TO TGenericStatusWord;
END_VAR
VAR
	wordSum: WORD;
	cnt: BYTE;
END_VAR

wordSum    := wordSum + SHL( BIT_TO_WORD( pBitPointer^.bit0 ) , 0 );
wordSum    := wordSum + SHL( BIT_TO_WORD( pBitPointer^.bit1 ) , 1 );
wordSum    := wordSum + SHL( BIT_TO_WORD( pBitPointer^.bit2 ) , 2 );
wordSum    := wordSum + SHL( BIT_TO_WORD( pBitPointer^.bit3 ) , 3 );
wordSum    := wordSum + SHL( BIT_TO_WORD( pBitPointer^.bit4 ) , 4 );
wordSum    := wordSum + SHL( BIT_TO_WORD( pBitPointer^.bit5 ) , 5 );
wordSum    := wordSum + SHL( BIT_TO_WORD( pBitPointer^.bit6 ) , 6 );
wordSum    := wordSum + SHL( BIT_TO_WORD( pBitPointer^.bit7 ) , 7 );
wordSum    := wordSum + SHL( BIT_TO_WORD( pBitPointer^.bit8 ) , 8 );
wordSum    := wordSum + SHL( BIT_TO_WORD( pBitPointer^.bit9 ) , 9 );
wordSum    := wordSum + SHL( BIT_TO_WORD( pBitPointer^.bit10 ) , 10 );
wordSum    := wordSum + SHL( BIT_TO_WORD( pBitPointer^.bit11 ) , 11 );
wordSum    := wordSum + SHL( BIT_TO_WORD( pBitPointer^.bit12 ) , 12 );
wordSum    := wordSum + SHL( BIT_TO_WORD( pBitPointer^.bit13 ) , 13 );
wordSum    := wordSum + SHL( BIT_TO_WORD( pBitPointer^.bit14 ) , 14 );
wordSum    := wordSum + SHL( BIT_TO_WORD( pBitPointer^.bit15 ) , 15 );

F_STATUS_WORD_TO_WORD    := wordSum;

END_FUNCTION

// 20 Program Organization Units/Utility Functions/fb_Clock
(*AUTHOR:			Jaison Schaab*)
(*DATE:				November 5 / 2019*)
(*DESCRIPTION: 		This Function Block will generate a clock signal based on defined ON/OFF times*)

(*UPDATE: 			March. 18 2021 - Jaison Schaab

					Code Ported from Wago.
					
					Code Is fully tested and functional.
*)

FUNCTION_BLOCK fb_Clock
VAR_INPUT
	xEnable 	: BOOL;		(* clock runs while this input true. *)
	tT_ON 		: TIME;		(* time while xOut is true *)
	tT_OFF 		: TIME;		(* time while xOut is false *)
END_VAR
VAR_OUTPUT
	xOut 		: BOOL;		(* clock output. Always true on startup *)
	xHstrobe 	: BOOL;		(* pulse on rising edge of xOut *)
	xLstrobe 	: BOOL;		(* pulse on falling edge of xOut *)
END_VAR
VAR
	off			: BOOL;
	on			: BOOL;
	mark		: BOOL;
	space		: BOOL;
	onTRIG		: F_TRIG;
	offTRIG		: F_TRIG;
	m			: TP;
	sp			: TP;
	kick		: R_TRIG;
	kk			: BOOL;
END_VAR

kick(CLK:=xEnable, Q=> kk);
IF xEnable = TRUE THEN
	ontrig(CLK:= space, Q=>on );
	m(IN:= on OR kk, PT:=tT_ON , Q=>mark);
	offtrig(CLK:= mark, Q=>off );
	sp(IN:= off, PT:=tT_OFF , Q=>space);
	xOut:= mark;
	xHstrobe := on;
	xLstrobe := off;
ELSE
	xOut:=FALSE;
END_IF;

END_FUNCTION_BLOCK

// 20 Program Organization Units/Utility Functions/fb_GetCycleTime
(*AUTHOR:		Jaison Schaab*)
(*DATE:			March. 11 / 2020*)
(*DESCRIPTION: 	This function block will report the PLC cycle time. *)
					
(*NOTES:		To be called every scan to report the program cycle time.

				This is a generic way to report the cycle time which is NOT
				tied to a local global veriable as was done in the previous
				program template.
*)

(*UPDATE: 			March. 18 2021 - Jaison Schaab

					Code Ported from Wago.
					
					Code Is fully tested and functional.
*)

(*UPDATE: 		June. 19 2020 - Jaison Schaab
					
				Fixed the 100ns output which is too large for a UINT so was
				getting truncated.  Needed to update it to be a ULINT.
*)

FUNCTION_BLOCK fb_GetCycleTime
VAR_INPUT
END_VAR
VAR_OUTPUT
	CycleTime_us		: UINT;					// Cycle Time of the PLC in microseconds (us)
	CycleTime_100ns		: ULINT; 				// Cycle Time of the PLC in 100 Nanoseconds (100 ns)
END_VAR
VAR
	CycleTimer			: fb_ElapsedTime;		// Elapsed time function block
END_VAR
VAR CONSTANT
	ns_TO_us_MULT		: LREAL := 0.001;		// nanoseconds to microseconds multiplier
	ns_TO_100ns_MULT	: LREAL := 0.01;		// nanoseconds to 100 nanoseconds multiplier
END_VAR

// Calculate the cycle time in Microseconds (us)
CycleTime_us := TO_UINT(TO_LREAL(CycleTimer.GetElapsedLTime()) * ns_TO_us_MULT);

// Calculate the cycle time in 100 Nanoseconds (100 ns)
CycleTime_100ns := TO_ULINT(TO_LREAL(CycleTimer.GetElapsedLTime()) * ns_TO_100ns_MULT);

// Reset the elapsed timer
CycleTimer.StartNow();

END_FUNCTION_BLOCK

// 20 Program Organization Units/Utility Functions/fb_TriggerTimer
(*AUTHOR:			Jaison Schaab*)
(*DATE:				November 26 / 2019*)
(*DESCRIPTION: 		This Function Block returns the elapsed time between rising edge triggers.*)

(*UPDATE: 			March. 18 2021 - Jaison Schaab

					Code Ported from Wago.
					
					Code Is fully tested and functional.
*)

(*UPDATE: 			March. 18 2021 - Jaison Schaab

					Code Ported from Wago.
					
					Through testing it was discovered that the TIME / LTIME variables and their
					conversion routines are handled differently.  Because of this I have renamed
					the output variables as well as the logic such that the timer values are correct.
*)

FUNCTION_BLOCK fb_TriggerTimer
VAR_INPUT
	xEnable					: BOOL;
	xTrigger				: BOOL;
END_VAR
VAR_OUTPUT
	tTrigger_Time			: TIME;			// Value for Round Trip Message Time
	tTrigger_LTime			: LTIME;		// Value for Round Trip Message LTime
	uiTrigger_Time_ms		: UINT;			// Value for Round Trip Message Time in milliseconds (ms)
END_VAR
VAR
	ValueChangeTrigger		: R_TRIG;
	TriggerTimer			: fb_ElapsedTime;
END_VAR

// Trigger a value changed event
ValueChangeTrigger(CLK:= xTrigger);

// Run the round trip timer
TriggerTimer();

IF xEnable THEN

	// Reset the timer whenever the value changed trigger is TRUE
	IF (ValueChangeTrigger.Q) THEN
	// Output the measured Round Trip Time
	tTrigger_Time		 := TriggerTimer.GetElapsedTime();
	tTrigger_LTime 		:= TriggerTimer.GetElapsedLTime();
	
	uiTrigger_Time_ms 	:= LTIME_TO_UINT(tTrigger_LTime / 1000000); 	// Sanity Check - Milliseconds
	
	// Reset the elapsed timer
	TriggerTimer.StartNow();
	
	END_IF

ELSE
		
	tTrigger_Time 		:= T#0S;
	tTrigger_LTime 		:= TIME_TO_LTIME(T#0S);
	uiTrigger_Time_ms 	:= 0;
	
END_IF

END_FUNCTION_BLOCK

// 20 Program Organization Units/Utility Functions/Logger
(*AUTHOR:		James Belcher*)
(*DATE:			 *)
(*DESCRIPTION:	This Function logs events that you want to be aware of.*)
(*
NOTES:  
INPUTS: index 		: UINT; 			// different indexes for different call of this function
		timestamp 	: TIME;				// Time stamp
		msg 		: STRING(20);		// Event message
		count 		: UINT;				// increasing count	   					
VAR_IN_OUTs:     				
FUNCTIONALITY: 			  
OUTPUTS:       
EXAMPLE CODE USAGE: event log usage on Frac Pumper: dataLogger.LogPoint( 1 , TO_TIME( gCycleTime_us * 1000 ) , 'COMM OK EVNT' , dataLogger.getCount( 1 ) + 1 );	
													dataLogger.LogPoint( 2 , TO_TIME( gCycleTime_us * 1000 ) , 'COMM LOSS EVNT' , dataLogger.getCount( 2 ) + 1 );	
*)
(*UPDATE: 		*)		

FUNCTION_BLOCK Logger
VAR_INPUT
END_VAR
VAR_OUTPUT
END_VAR
VAR
	dataPoints : ARRAY [1..20] OF DataPoint;
END_VAR

METHOD getCount : UINT
VAR_INPUT
	index: UINT;
END_VAR
getCount := dataPoints[index].counter;
END_METHOD

METHOD LogPoint
VAR_INPUT
	index: UINT;
	timestamp: TIME;
	msg: STRING(20);
	count: UINT;
END_VAR
dataPoints[index].timestamp := timestamp;
dataPoints[index].message := msg;
dataPoints[index].counter := count;
END_METHOD

END_FUNCTION_BLOCK

// Project Information/F_GetCompany
// This function has been automatically generated from the project information.
{attribute 'signature_flag' := '1073741824'}
{attribute 'TcGenerated'}
{attribute 'no-analysis'}
FUNCTION F_GetCompany : WSTRING
VAR_INPUT
	
END_VAR

F_GetCompany := "National Oilwell Varco";

END_FUNCTION

// Project Information/F_GetTitle
// This function has been automatically generated from the project information.
{attribute 'signature_flag' := '1073741824'}
{attribute 'TcGenerated'}
{attribute 'no-analysis'}
FUNCTION F_GetTitle : WSTRING
VAR_INPUT
	
END_VAR

F_GetTitle := "stdNOV";

END_FUNCTION

// Project Information/F_GetVersion
// This function has been automatically generated from the project information.
{attribute 'signature_flag' := '1073741824'}
{attribute 'TcGenerated'}
{attribute 'no-analysis'}
FUNCTION F_GetVersion : ST_LibVersion
VAR_INPUT
	
END_VAR

F_GetVersion.iMajor := 1;
F_GetVersion.iMinor := 0;
F_GetVersion.iBuild := 0;
F_GetVersion.iRevision := 2936;

END_FUNCTION
